C03619=1072.595,223.808,-82.460,174.049,27.815,154.953
C03620=1072.590,223.559,-82.434,174.047,27.812,154.952
C03621=1072.583,223.310,-82.409,174.044,27.808,154.952
C03622=1072.578,223.061,-82.383,174.043,27.804,154.951
C03623=1072.572,222.850,-82.361,174.041,27.800,154.951
C03624=1072.568,222.638,-82.338,174.039,27.797,154.950
C03625=1072.563,222.426,-82.317,174.037,27.794,154.949
C03626=1072.558,222.213,-82.294,174.035,27.790,154.949
C03627=1072.553,222.002,-82.272,174.033,27.787,154.948
C03628=1072.548,221.790,-82.250,174.032,27.784,154.948
C03629=1072.543,221.577,-82.228,174.030,27.780,154.947
C03630=1072.538,221.365,-82.207,174.028,27.777,154.947
C03631=1072.533,221.116,-82.181,174.025,27.773,154.946
C03632=1072.526,220.868,-82.155,174.023,27.769,154.946
C03633=1072.520,220.619,-82.129,174.022,27.766,154.945
C03634=1072.515,220.371,-82.104,174.019,27.761,154.944
C03635=1072.509,220.122,-82.078,174.017,27.758,154.944
C03636=1072.503,219.873,-82.052,174.015,27.754,154.943
C03637=1072.497,219.625,-82.027,174.012,27.750,154.943
C03638=1072.491,219.377,-82.001,174.010,27.746,154.942
C03639=1072.485,219.128,-81.975,174.009,27.743,154.941
C03640=1072.479,218.879,-81.950,174.006,27.738,154.941
C03641=1072.473,218.630,-81.924,174.004,27.734,154.940
C03642=1072.468,218.382,-81.899,174.002,27.731,154.940
C03643=1072.462,218.133,-81.873,173.999,27.727,154.939
C03644=1072.456,217.885,-81.848,173.998,27.723,154.938
C03645=1072.450,217.636,-81.822,173.996,27.719,154.938
C03646=1072.444,217.387,-81.796,173.994,27.715,154.937
C03647=1072.439,217.139,-81.771,173.991,27.711,154.936
C03648=1072.433,216.890,-81.746,173.989,27.707,154.936
C03649=1072.427,216.641,-81.720,173.987,27.703,154.935
C03650=1072.421,216.393,-81.695,173.985,27.699,154.935
C03651=1072.415,216.144,-81.669,173.983,27.695,154.934
C03652=1072.410,215.896,-81.644,173.981,27.692,154.933
C03653=1072.404,215.647,-81.618,173.978,27.688,154.933
C03654=1072.398,215.398,-81.593,173.976,27.684,154.932
C03655=1072.392,215.149,-81.567,173.975,27.680,154.931
C03656=1072.386,214.901,-81.542,173.972,27.676,154.931
C03657=1072.381,214.652,-81.518,173.970,27.672,154.930
C03658=1072.375,214.403,-81.492,173.968,27.668,154.930
C03659=1072.369,214.154,-81.466,173.965,27.664,154.929
C03660=1072.363,213.906,-81.441,173.964,27.660,154.928
C03661=1072.358,213.657,-81.415,173.962,27.656,154.928
C03662=1072.352,213.409,-81.390,173.960,27.652,154.927
C03663=1072.346,213.161,-81.365,173.957,27.648,154.926
C03664=1072.340,212.912,-81.340,173.956,27.645,154.926
C03665=1072.335,212.663,-81.315,173.954,27.641,154.925
C03666=1072.328,212.414,-81.289,173.951,27.637,154.925
C03667=1072.323,212.166,-81.264,173.949,27.633,154.924
C03668=1072.317,211.917,-81.240,173.947,27.629,154.923
C03669=1072.311,211.668,-81.214,173.945,27.625,154.923
C03670=1072.306,211.420,-81.189,173.943,27.621,154.922
C03671=1072.300,211.171,-81.163,173.941,27.617,154.922
C03672=1072.294,210.922,-81.139,173.939,27.613,154.921
C03673=1072.288,210.673,-81.113,173.937,27.609,154.920
C03674=1072.282,210.425,-81.088,173.935,27.606,154.920
C03675=1072.276,210.176,-81.064,173.933,27.602,154.919
C03676=1072.270,209.927,-81.038,173.930,27.598,154.918
C03677=1072.264,209.679,-81.013,173.928,27.593,154.918
C03678=1072.258,209.430,-80.989,173.927,27.590,154.917
C03679=1072.249,209.010,-80.946,173.923,27.583,154.916
C03680=1072.239,208.591,-80.904,173.919,27.577,154.915
C03681=1072.229,208.171,-80.862,173.916,27.570,154.914
C03682=1072.220,207.751,-80.820,173.912,27.563,154.913
C03683=1072.195,206.710,-80.719,173.782,27.496,154.911
C03684=1072.190,206.461,-80.694,173.780,27.493,154.911
C03685=1072.184,206.212,-80.670,173.778,27.490,154.911
C03686=1072.178,205.964,-80.646,173.776,27.487,154.910
C03687=1072.173,205.715,-80.622,173.773,27.484,154.910
C03688=1072.167,205.466,-80.597,173.771,27.480,154.909
C03689=1072.161,205.217,-80.573,173.769,27.477,154.909
C03690=1072.155,204.969,-80.549,173.767,27.475,154.909
C03691=1072.150,204.720,-80.525,173.765,27.472,154.908
C03692=1072.144,204.471,-80.500,173.762,27.469,154.908
C03693=1072.139,204.222,-80.476,173.760,27.465,154.907
C03694=1072.133,203.974,-80.452,173.758,27.463,154.907
C03695=1072.127,203.724,-80.428,173.756,27.460,154.907
C03696=1072.122,203.476,-80.404,173.753,27.457,154.906
C03697=1072.116,203.227,-80.381,173.751,27.454,154.906
C03698=1072.111,202.979,-80.356,173.749,27.451,154.905
C03699=1072.105,202.729,-80.332,173.747,27.448,154.905
C03700=1072.099,202.481,-80.307,173.745,27.444,154.905
C03701=1072.094,202.232,-80.284,173.742,27.441,154.904
C03702=1072.088,201.983,-80.260,173.741,27.439,154.904
C03703=1072.082,201.734,-80.236,173.738,27.436,154.903
C03704=1072.076,201.486,-80.212,173.736,27.433,154.903
C03705=1072.070,201.238,-80.188,173.733,27.430,154.903
C03706=1072.065,200.988,-80.164,173.732,27.427,154.902
C03707=1072.059,200.739,-80.141,173.729,27.424,154.902
C03708=1072.053,200.491,-80.117,173.727,27.421,154.902
C03709=1072.047,200.241,-80.093,173.724,27.418,154.901
C03710=1072.041,199.993,-80.069,173.723,27.416,154.901
C03711=1072.036,199.744,-80.045,173.720,27.413,154.900
C03712=1072.030,199.495,-80.022,173.718,27.410,154.900
C03713=1072.024,199.246,-79.998,173.716,27.407,154.900
C03714=1072.018,198.998,-79.974,173.714,27.404,154.899
C03715=1072.013,198.749,-79.950,173.712,27.401,154.899
C03716=1072.007,198.500,-79.927,173.709,27.398,154.898
C03717=1072.001,198.251,-79.903,173.707,27.395,154.898
C03718=1071.996,198.002,-79.879,173.705,27.393,154.898
C03719=1071.989,197.754,-79.856,173.703,27.390,154.897
C03720=1071.984,197.505,-79.832,173.700,27.387,154.897
C03721=1071.978,197.256,-79.808,173.699,27.384,154.897
C03722=1071.972,197.007,-79.784,173.696,27.381,154.896
C03723=1071.967,196.758,-79.761,173.694,27.378,154.896
C03724=1071.961,196.510,-79.737,173.692,27.375,154.895
C03725=1071.956,196.261,-79.714,173.690,27.372,154.895
C03726=1071.950,196.012,-79.690,173.688,27.369,154.895
C03727=1071.943,195.763,-79.667,173.685,27.366,154.894
C03728=1071.938,195.514,-79.642,173.684,27.364,154.894
C03729=1071.932,195.265,-79.619,173.681,27.361,154.893
C03730=1071.927,195.017,-79.595,173.679,27.358,154.893
C03731=1071.921,194.768,-79.572,173.677,27.355,154.893
C03732=1071.915,194.520,-79.549,173.675,27.352,154.892
C03733=1071.910,194.270,-79.525,173.672,27.349,154.892
C03734=1071.904,194.021,-79.501,173.671,27.346,154.892
C03735=1071.898,193.773,-79.478,173.668,27.343,154.891
C03736=1071.893,193.523,-79.454,173.666,27.340,154.891
C03737=1071.887,193.275,-79.431,173.664,27.337,154.890
C03738=1071.881,193.026,-79.408,173.662,27.334,154.890
C03739=1071.876,192.778,-79.384,173.660,27.331,154.890
C03740=1071.870,192.529,-79.361,173.658,27.328,154.889
C03741=1071.864,192.280,-79.338,173.656,27.325,154.889
C03742=1071.859,192.031,-79.313,173.653,27.323,154.888
C03743=1071.853,191.782,-79.291,173.652,27.320,154.888
C03744=1071.847,191.501,-79.264,173.649,27.317,154.888
C03745=1071.841,191.219,-79.238,173.647,27.314,154.887
C03746=1071.834,190.938,-79.211,173.645,27.310,154.887
C03747=1071.828,190.656,-79.184,173.642,27.307,154.886
C03748=1071.822,190.407,-79.161,173.640,27.304,154.886
C03749=1071.817,190.158,-79.138,173.637,27.301,154.886
C03750=1071.811,189.909,-79.115,173.636,27.298,154.885
C03751=1071.805,189.661,-79.091,173.633,27.295,154.885
C03752=1071.800,189.411,-79.068,173.631,27.292,154.884
C03753=1071.795,189.162,-79.045,173.629,27.289,154.884
C03754=1071.789,188.914,-79.022,173.627,27.286,154.884
C03755=1071.783,188.665,-78.998,173.625,27.283,154.883
C03756=1071.778,188.416,-78.975,173.623,27.281,154.883
C03757=1071.772,188.167,-78.952,173.621,27.278,154.882
C03758=1071.766,187.918,-78.929,173.619,27.275,154.882
C03759=1071.761,187.669,-78.905,173.617,27.272,154.882
C03760=1071.755,187.421,-78.881,173.614,27.269,154.881
C03761=1071.750,187.172,-78.859,173.613,27.267,154.881
C03762=1071.744,186.923,-78.836,173.610,27.263,154.881
C03763=1071.739,186.674,-78.812,173.608,27.260,154.880
C03764=1071.733,186.425,-78.789,173.606,27.258,154.880
C03765=1071.728,186.176,-78.766,173.604,27.255,154.879
C03766=1071.722,185.927,-78.743,173.602,27.252,154.879
C03767=1071.717,185.678,-78.720,173.600,27.249,154.879
C03768=1071.711,185.429,-78.697,173.598,27.246,154.878
C03769=1071.705,185.180,-78.674,173.596,27.243,154.878
C03770=1071.700,184.931,-78.651,173.594,27.240,154.877
C03771=1071.694,184.683,-78.628,173.592,27.237,154.877
C03772=1071.688,184.433,-78.605,173.590,27.234,154.877
C03773=1071.682,184.185,-78.582,173.587,27.232,154.876
C03774=1071.677,183.936,-78.559,173.586,27.229,154.876
C03775=1071.671,183.687,-78.536,173.583,27.226,154.875
C03776=1071.665,183.438,-78.513,173.582,27.224,154.875
C03777=1071.659,183.189,-78.490,173.579,27.221,154.875
C03778=1071.653,182.940,-78.468,173.577,27.218,154.874
C03779=1071.647,182.691,-78.445,173.575,27.215,154.874
C03780=1071.642,182.443,-78.422,173.573,27.212,154.874
C03781=1071.636,182.194,-78.399,173.571,27.210,154.873
C03782=1071.630,181.945,-78.376,173.569,27.207,154.873
C03783=1071.624,181.696,-78.354,173.567,27.204,154.873
C03784=1071.618,181.447,-78.331,173.565,27.201,154.872
C03785=1071.612,181.198,-78.309,173.563,27.198,154.872
C03786=1071.607,180.949,-78.286,173.561,27.196,154.872
C03787=1071.602,180.701,-78.263,173.559,27.193,154.871
C03788=1071.595,180.452,-78.241,173.557,27.190,154.871
C03789=1071.589,180.203,-78.218,173.555,27.188,154.871
C03790=1071.584,179.954,-78.195,173.552,27.185,154.870
C03791=1071.578,179.705,-78.173,173.551,27.182,154.870
C03792=1071.573,179.456,-78.150,173.548,27.179,154.869
C03793=1071.566,179.207,-78.127,173.547,27.177,154.869
C03794=1071.560,178.958,-78.104,173.544,27.174,154.869
C03795=1071.555,178.709,-78.081,173.543,27.171,154.868
C03796=1071.549,178.460,-78.059,173.540,27.168,154.868
C03797=1071.543,178.211,-78.037,173.539,27.166,154.868
C03798=1071.537,177.962,-78.014,173.536,27.163,154.867
C03799=1071.532,177.714,-77.992,173.534,27.160,154.867
C03800=1071.526,177.465,-77.969,173.532,27.157,154.867
C03801=1071.520,177.216,-77.947,173.530,27.154,154.866
C03802=1071.514,176.967,-77.924,173.529,27.152,154.866
C03803=1071.509,176.718,-77.902,173.526,27.148,154.865
C03804=1071.503,176.469,-77.879,173.525,27.146,154.865
C03805=1071.497,176.220,-77.856,173.522,27.143,154.865
C03806=1071.492,175.971,-77.834,173.521,27.140,154.864
C03807=1071.486,175.723,-77.811,173.518,27.137,154.864
C03808=1071.479,175.441,-77.786,173.516,27.134,154.864
C03809=1071.473,175.158,-77.761,173.513,27.131,154.863
C03810=1071.466,174.877,-77.735,173.512,27.129,154.863
C03811=1071.460,174.595,-77.710,173.510,27.125,154.862
C03812=1071.454,174.345,-77.688,173.507,27.122,154.862
C03813=1071.448,174.096,-77.665,173.506,27.120,154.862
C03814=1071.444,173.847,-77.643,173.503,27.117,154.861
C03815=1071.437,173.599,-77.620,173.502,27.114,154.861
C03816=1071.431,173.350,-77.597,173.499,27.111,154.861
C03817=1071.426,173.100,-77.575,173.498,27.109,154.860
C03818=1071.420,172.852,-77.553,173.495,27.106,154.860
C03819=1071.415,172.603,-77.531,173.494,27.103,154.859
C03820=1071.409,172.354,-77.508,173.491,27.100,154.859
C03821=1071.403,172.105,-77.486,173.490,27.097,154.859
C03822=1071.398,171.857,-77.464,173.488,27.094,154.858
C03823=1071.392,171.607,-77.442,173.486,27.092,154.858
C03824=1071.386,171.359,-77.419,173.484,27.089,154.858
C03825=1071.380,171.109,-77.397,173.482,27.086,154.857
C03826=1071.375,170.860,-77.375,173.480,27.083,154.857
C03827=1071.369,170.612,-77.353,173.478,27.081,154.856
C03828=1071.364,170.362,-77.331,173.476,27.078,154.856
C03829=1071.358,170.113,-77.308,173.474,27.075,154.856
C03830=1071.352,169.865,-77.286,173.472,27.072,154.855
C03831=1071.347,169.616,-77.263,173.470,27.069,154.855
C03832=1071.341,169.366,-77.241,173.468,27.066,154.855
C03833=1071.336,169.118,-77.220,173.466,27.064,154.854
C03834=1071.330,168.869,-77.197,173.464,27.061,154.854
C03835=1071.324,168.619,-77.175,173.463,27.058,154.853
C03836=1071.319,168.371,-77.154,173.460,27.055,154.853
C03837=1071.313,168.122,-77.131,173.459,27.052,154.853
C03838=1071.308,167.872,-77.108,173.456,27.050,154.852
C03839=1071.302,167.624,-77.087,173.455,27.047,154.852
C03840=1071.296,167.375,-77.064,173.452,27.044,154.852
C03841=1071.290,167.126,-77.042,173.451,27.041,154.851
C03842=1071.285,166.877,-77.021,173.448,27.038,154.851
C03843=1071.280,166.628,-76.998,173.447,27.036,154.851
C03844=1071.274,166.380,-76.976,173.445,27.033,154.850
C03845=1071.269,166.130,-76.954,173.443,27.030,154.850
C03846=1071.263,165.881,-76.933,173.442,27.027,154.849
C03847=1071.258,165.632,-76.911,173.439,27.024,154.849
C03848=1071.252,165.383,-76.888,173.438,27.022,154.849
C03849=1071.246,165.135,-76.866,173.435,27.019,154.848
C03850=1071.241,164.885,-76.844,173.434,27.016,154.848
C03851=1071.235,164.636,-76.823,173.431,27.013,154.848
C03852=1071.230,164.387,-76.801,173.430,27.010,154.847
C03853=1071.224,164.138,-76.778,173.428,27.008,154.847
C03854=1071.219,163.890,-76.757,173.426,27.005,154.846
C03855=1071.213,163.640,-76.734,173.424,27.002,154.846
C03856=1071.208,163.392,-76.713,173.422,26.999,154.846
C03857=1071.202,163.142,-76.691,173.421,26.997,154.845
C03858=1071.197,162.894,-76.670,173.418,26.994,154.845
C03859=1071.191,162.645,-76.647,173.417,26.991,154.844
C03860=1071.186,162.395,-76.624,173.415,26.988,154.844
C03861=1071.180,162.147,-76.603,173.413,26.985,154.844
C03862=1071.175,161.897,-76.581,173.411,26.983,154.843
C03863=1071.169,161.649,-76.560,173.409,26.980,154.843
C03864=1071.164,161.399,-76.537,173.407,26.977,154.843
C03865=1071.158,161.151,-76.516,173.405,26.974,154.842
C03866=1071.152,160.902,-76.494,173.403,26.972,154.842
C03867=1071.147,160.653,-76.473,173.402,26.969,154.841
C03868=1071.141,160.404,-76.451,173.400,26.966,154.841
C03869=1071.135,160.154,-76.429,173.398,26.963,154.841
C03870=1071.129,159.906,-76.408,173.396,26.960,154.840
C03871=1071.124,159.656,-76.386,173.394,26.958,154.840
C03872=1071.117,159.374,-76.361,173.392,26.955,154.840
C03873=1071.111,159.092,-76.337,173.389,26.951,154.839
C03874=1071.104,158.810,-76.313,173.388,26.949,154.839
C03875=1071.098,158.527,-76.289,173.386,26.946,154.838
C03876=1071.092,158.278,-76.266,173.384,26.943,154.838
C03877=1071.087,158.029,-76.245,173.382,26.940,154.838
C03878=1071.080,157.780,-76.224,173.380,26.937,154.837
C03879=1071.075,157.531,-76.202,173.378,26.934,154.837
C03880=1071.069,157.282,-76.180,173.376,26.932,154.837
C03881=1071.064,157.033,-76.159,173.375,26.929,154.836
C03882=1071.058,156.784,-76.137,173.372,26.926,154.836
C03883=1071.052,156.535,-76.117,173.371,26.924,154.836
C03884=1071.046,156.286,-76.095,173.369,26.920,154.835
C03885=1071.042,156.037,-76.073,173.367,26.918,154.835
C03886=1071.035,155.788,-76.051,173.366,26.915,154.834
C03887=1071.030,155.539,-76.030,173.363,26.912,154.834
C03888=1071.024,155.290,-76.009,173.362,26.910,154.834
C03889=1071.018,155.041,-75.988,173.359,26.907,154.833
C03890=1071.012,154.792,-75.966,173.358,26.904,154.833
C03891=1071.007,154.543,-75.945,173.356,26.902,154.833
C03892=1071.000,154.294,-75.923,173.354,26.899,154.832
C03893=1070.996,154.045,-75.902,173.352,26.896,154.832
C03894=1070.990,153.795,-75.881,173.351,26.893,154.832
C03895=1070.984,153.547,-75.859,173.348,26.891,154.831
C03896=1070.978,153.298,-75.838,173.347,26.888,154.831
C03897=1070.973,153.049,-75.817,173.345,26.885,154.830
C03898=1070.967,152.799,-75.796,173.343,26.883,154.830
C03899=1070.961,152.551,-75.774,173.342,26.880,154.830
C03900=1070.955,152.302,-75.753,173.339,26.877,154.829
C03901=1070.950,152.053,-75.732,173.338,26.875,154.829
C03902=1070.944,151.804,-75.711,173.336,26.872,154.829
C03903=1070.938,151.555,-75.689,173.334,26.869,154.828
C03904=1070.933,151.306,-75.669,173.332,26.866,154.828
C03905=1070.927,151.056,-75.647,173.331,26.864,154.828
C03906=1070.921,150.808,-75.626,173.328,26.861,154.827
C03907=1070.915,150.558,-75.605,173.327,26.858,154.827
C03908=1070.910,150.310,-75.584,173.324,26.855,154.827
C03909=1070.904,150.061,-75.563,173.323,26.853,154.826
C03910=1070.898,149.811,-75.541,173.322,26.850,154.826
C03911=1070.893,149.563,-75.520,173.319,26.847,154.826
C03912=1070.887,149.313,-75.499,173.318,26.844,154.825
C03913=1070.881,149.064,-75.478,173.316,26.842,154.825
C03914=1070.876,148.815,-75.457,173.314,26.839,154.824
C03915=1070.870,148.566,-75.436,173.312,26.836,154.824
C03916=1070.864,148.317,-75.415,173.311,26.834,154.824
C03917=1070.858,148.068,-75.394,173.308,26.830,154.823
C03918=1070.853,147.819,-75.373,173.307,26.828,154.823
C03919=1070.847,147.570,-75.352,173.305,26.825,154.823
C03920=1070.842,147.320,-75.331,173.303,26.823,154.822
C03921=1070.836,147.072,-75.310,173.301,26.820,154.822
C03922=1070.829,146.822,-75.289,173.300,26.817,154.821
C03923=1070.824,146.574,-75.268,173.298,26.815,154.821
C03924=1070.819,146.325,-75.247,173.296,26.812,154.821
C03925=1070.813,146.076,-75.226,173.295,26.809,154.820
C03926=1070.807,145.826,-75.205,173.292,26.807,154.820
C03927=1070.802,145.578,-75.184,173.291,26.804,154.820
C03928=1070.795,145.328,-75.164,173.289,26.801,154.819
C03929=1070.790,145.079,-75.143,173.287,26.799,154.819
C03930=1070.784,144.830,-75.121,173.285,26.796,154.819
C03931=1070.778,144.581,-75.101,173.284,26.793,154.818
C03932=1070.773,144.332,-75.080,173.281,26.790,154.818
C03933=1070.766,144.083,-75.059,173.280,26.788,154.818
C03934=1070.761,143.834,-75.039,173.279,26.785,154.817
C03935=1070.755,143.585,-75.017,173.276,26.782,154.817
C03936=1070.749,143.302,-74.994,173.275,26.779,154.816
C03937=1070.742,143.020,-74.970,173.272,26.776,154.816
C03938=1070.736,142.737,-74.947,173.271,26.773,154.816
C03939=1070.729,142.455,-74.923,173.269,26.770,154.815
C03940=1070.724,142.205,-74.902,173.267,26.767,154.815
C03941=1070.718,141.956,-74.882,173.265,26.765,154.815
C03942=1070.712,141.707,-74.861,173.263,26.762,154.814
C03943=1070.707,141.458,-74.840,173.262,26.759,154.814
C03944=1070.702,141.209,-74.820,173.259,26.756,154.813
C03945=1070.696,140.959,-74.799,173.258,26.754,154.813
C03946=1070.689,140.711,-74.778,173.256,26.751,154.813
C03947=1070.684,140.462,-74.758,173.255,26.748,154.812
C03948=1070.679,140.213,-74.737,173.252,26.746,154.812
C03949=1070.672,139.963,-74.717,173.251,26.743,154.812
C03950=1070.667,139.715,-74.695,173.250,26.740,154.811
C03951=1070.661,139.466,-74.675,173.247,26.737,154.811
C03952=1070.655,139.216,-74.655,173.246,26.735,154.811
C03953=1070.650,138.967,-74.634,173.244,26.732,154.810
C03954=1070.644,138.718,-74.613,173.243,26.730,154.810
C03955=1070.638,138.469,-74.593,173.240,26.726,154.809
C03956=1070.632,138.220,-74.572,173.239,26.724,154.809
C03957=1070.626,137.971,-74.552,173.237,26.721,154.809
C03958=1070.621,137.722,-74.531,173.235,26.718,154.808
C03959=1070.616,137.473,-74.511,173.234,26.716,154.808
C03960=1070.609,137.223,-74.490,173.232,26.713,154.808
C03961=1070.604,136.974,-74.470,173.231,26.710,154.807
C03962=1070.598,136.725,-74.450,173.228,26.707,154.807
C03963=1070.593,136.476,-74.429,173.227,26.705,154.807
C03964=1070.586,136.227,-74.408,173.225,26.702,154.806
C03965=1070.580,135.978,-74.388,173.223,26.699,154.806
C03966=1070.575,135.729,-74.367,173.221,26.697,154.806
C03967=1070.569,135.480,-74.347,173.220,26.694,154.805
C03968=1070.564,135.231,-74.327,173.218,26.691,154.805
C03969=1070.557,134.982,-74.306,173.216,26.689,154.805
C03970=1070.552,134.733,-74.286,173.215,26.686,154.804
C03971=1070.546,134.484,-74.266,173.213,26.683,154.804
C03972=1070.541,134.235,-74.245,173.212,26.681,154.803
C03973=1070.535,133.986,-74.225,173.209,26.678,154.803
C03974=1070.529,133.736,-74.204,173.208,26.675,154.803
C03975=1070.523,133.487,-74.185,173.206,26.673,154.802
C03976=1070.518,133.238,-74.164,173.205,26.670,154.802
C03977=1070.512,132.989,-74.144,173.202,26.667,154.802
C03978=1070.506,132.740,-74.123,173.201,26.665,154.801
C03979=1070.500,132.491,-74.103,173.199,26.662,154.801
C03980=1070.495,132.242,-74.083,173.198,26.659,154.800
C03981=1070.489,131.992,-74.063,173.196,26.656,154.800
C03982=1070.484,131.743,-74.043,173.194,26.654,154.800
C03983=1070.478,131.494,-74.023,173.193,26.651,154.799
C03984=1070.472,131.245,-74.003,173.191,26.649,154.799
C03985=1070.466,130.996,-73.982,173.189,26.646,154.799
C03986=1070.460,130.747,-73.962,173.187,26.643,154.798
C03987=1070.454,130.498,-73.942,173.186,26.640,154.798
C03988=1070.448,130.249,-73.922,173.184,26.638,154.798
C03989=1070.443,129.999,-73.902,173.182,26.635,154.797
C03990=1070.437,129.751,-73.882,173.180,26.632,154.797
C03991=1070.430,129.501,-73.862,173.179,26.630,154.797
C03992=1070.424,129.252,-73.842,173.178,26.627,154.796
C03993=1070.419,129.003,-73.821,173.175,26.624,154.796
C03994=1070.413,128.754,-73.802,173.174,26.622,154.796
C03995=1070.407,128.505,-73.782,173.172,26.619,154.795
C03996=1070.401,128.256,-73.762,173.171,26.617,154.795
C03997=1070.396,128.006,-73.741,173.168,26.614,154.795
C03998=1070.390,127.757,-73.721,173.167,26.611,154.794
C03999=1070.384,127.508,-73.702,173.165,26.609,154.794
C04000=1070.378,127.226,-73.679,173.163,26.606,154.793
C04001=1070.371,126.943,-73.656,173.162,26.602,154.793
C04002=1070.364,126.660,-73.634,173.159,26.599,154.793
C04003=1070.358,126.377,-73.611,173.158,26.596,154.792
C04004=1070.352,126.128,-73.591,173.156,26.594,154.792
C04005=1070.346,125.879,-73.572,173.154,26.591,154.792
C04006=1070.340,125.630,-73.552,173.153,26.588,154.791
C04007=1070.335,125.380,-73.532,173.151,26.586,154.791
C04008=1070.329,125.132,-73.512,173.150,26.583,154.790
C04009=1070.323,124.883,-73.492,173.148,26.580,154.790
C04010=1070.317,124.633,-73.473,173.146,26.578,154.790
C04011=1070.311,124.385,-73.453,173.144,26.575,154.789
C04012=1070.306,124.134,-73.432,173.143,26.572,154.789
C04013=1070.300,123.885,-73.412,173.141,26.570,154.789
C04014=1070.294,123.636,-73.392,173.140,26.567,154.788
C04015=1070.288,123.387,-73.373,173.138,26.564,154.788
C04016=1070.282,123.138,-73.353,173.136,26.562,154.788
C04017=1070.277,122.888,-73.333,173.135,26.559,154.787
C04018=1070.271,122.640,-73.313,173.133,26.556,154.787
C04019=1070.265,122.391,-73.294,173.131,26.553,154.787
C04020=1070.260,122.141,-73.274,173.129,26.551,154.786
C04021=1070.254,121.893,-73.254,173.128,26.548,154.786
C04022=1070.248,121.643,-73.235,173.126,26.545,154.785
C04023=1070.243,121.394,-73.215,173.125,26.543,154.785
C04024=1070.237,121.145,-73.195,173.123,26.540,154.785
C04025=1070.231,120.896,-73.175,173.121,26.537,154.784
C04026=1070.225,120.646,-73.156,173.120,26.534,154.784
C04027=1070.219,120.398,-73.136,173.118,26.532,154.784
C04028=1070.214,120.148,-73.117,173.117,26.529,154.783
C04029=1070.208,119.899,-73.096,173.115,26.526,154.783
C04030=1070.203,119.650,-73.077,173.113,26.523,154.782
C04031=1070.197,119.401,-73.057,173.112,26.521,154.782
C04032=1070.191,119.151,-73.038,173.110,26.518,154.782
C04033=1070.185,118.903,-73.018,173.109,26.516,154.781
C04034=1070.180,118.654,-72.999,173.107,26.513,154.781
C04035=1070.174,118.405,-72.979,173.105,26.510,154.781
C04036=1070.168,118.156,-72.960,173.103,26.507,154.780
C04037=1070.163,117.906,-72.940,173.102,26.505,154.780
C04038=1070.157,117.657,-72.920,173.100,26.502,154.780
C04039=1070.151,117.408,-72.901,173.099,26.499,154.779
C04040=1070.146,117.159,-72.881,173.098,26.496,154.779
C04041=1070.140,116.909,-72.862,173.095,26.493,154.778
C04042=1070.134,116.660,-72.842,173.094,26.491,154.778
C04043=1070.128,116.411,-72.822,173.092,26.488,154.778
C04044=1070.122,116.162,-72.803,173.091,26.485,154.777
C04045=1070.117,115.912,-72.783,173.090,26.482,154.777
C04046=1070.112,115.664,-72.764,173.087,26.480,154.777
C04047=1070.106,115.414,-72.744,173.086,26.477,154.776
C04048=1070.101,115.165,-72.725,173.084,26.474,154.776
C04049=1070.095,114.916,-72.705,173.083,26.471,154.775
C04050=1070.089,114.667,-72.686,173.081,26.469,154.775
C04051=1070.083,114.417,-72.667,173.080,26.466,154.775
C04052=1070.077,114.168,-72.647,173.078,26.463,154.774
C04053=1070.072,113.919,-72.628,173.076,26.460,154.774
C04054=1070.067,113.670,-72.609,173.075,26.458,154.774
C04055=1070.061,113.421,-72.589,173.073,26.455,154.773
C04056=1070.055,113.172,-72.569,173.072,26.452,154.773
C04057=1070.049,112.923,-72.550,173.070,26.450,154.773
C04058=1070.043,112.673,-72.532,173.069,26.447,154.772
C04059=1070.037,112.424,-72.512,173.066,26.444,154.772
C04060=1070.031,112.175,-72.493,173.065,26.442,154.771
C04061=1070.025,111.926,-72.473,173.064,26.439,154.771
C04062=1070.020,111.676,-72.454,173.062,26.436,154.771
C04063=1070.015,111.428,-72.435,173.061,26.433,154.770
C04064=1070.007,111.144,-72.413,173.058,26.430,154.770
C04065=1070.001,110.861,-72.391,173.057,26.427,154.769
C04066=1069.995,110.579,-72.370,173.055,26.424,154.769
C04067=1069.988,110.297,-72.348,173.053,26.421,154.769
C04068=1069.982,110.047,-72.329,173.052,26.419,154.768
C04069=1069.976,109.798,-72.309,173.050,26.416,154.768
C04070=1069.970,109.549,-72.291,173.048,26.413,154.768
C04071=1069.964,109.299,-72.272,173.047,26.410,154.767
C04072=1069.959,109.050,-72.252,173.045,26.408,154.767
C04073=1069.953,108.800,-72.233,173.044,26.405,154.767
C04074=1069.946,108.551,-72.214,173.042,26.402,154.766
C04075=1069.941,108.303,-72.196,173.041,26.400,154.766
C04076=1069.936,108.053,-72.176,173.039,26.397,154.765
C04077=1069.930,107.804,-72.157,173.037,26.394,154.765
C04078=1069.924,107.555,-72.138,173.035,26.392,154.765
C04079=1069.918,107.305,-72.119,173.034,26.389,154.764
C04080=1069.912,107.056,-72.100,173.033,26.386,154.764
C04081=1069.906,106.807,-72.082,173.031,26.383,154.764
C04082=1069.901,106.558,-72.062,173.030,26.381,154.763
C04083=1069.895,106.308,-72.043,173.028,26.378,154.763
C04084=1069.889,106.059,-72.024,173.026,26.375,154.763
C04085=1069.883,105.810,-72.005,173.024,26.373,154.762
C04086=1069.878,105.561,-71.986,173.023,26.370,154.762
C04087=1069.872,105.312,-71.967,173.022,26.367,154.761
C04088=1069.866,105.063,-71.948,173.020,26.364,154.761
C04089=1069.860,104.813,-71.929,173.019,26.362,154.761
C04090=1069.854,104.564,-71.910,173.017,26.359,154.760
C04091=1069.848,104.315,-71.892,173.016,26.356,154.760
C04092=1069.843,104.066,-71.872,173.013,26.354,154.760
C04093=1069.837,103.816,-71.853,173.012,26.351,154.759
C04094=1069.831,103.567,-71.835,173.011,26.348,154.759
C04095=1069.826,103.319,-71.816,173.009,26.345,154.758
C04096=1069.820,103.069,-71.796,173.008,26.343,154.758
C04097=1069.814,102.820,-71.777,173.006,26.340,154.758
C04098=1069.808,102.570,-71.759,173.005,26.337,154.757
C04099=1069.803,102.321,-71.740,173.004,26.335,154.757
C04100=1069.797,102.072,-71.721,173.001,26.332,154.757
C04101=1069.791,101.823,-71.702,173.000,26.329,154.756
C04102=1069.786,101.574,-71.684,172.998,26.326,154.756
C04103=1069.779,101.325,-71.665,172.997,26.324,154.755
C04104=1069.774,101.075,-71.646,172.995,26.321,154.755
C04105=1069.768,100.825,-71.627,172.994,26.318,154.755
C04106=1069.762,100.577,-71.609,172.993,26.316,154.754
C04107=1069.757,100.328,-71.590,172.991,26.313,154.754
C04108=1069.750,100.078,-71.571,172.989,26.310,154.754
C04109=1069.744,99.829,-71.553,172.987,26.307,154.753
C04110=1069.739,99.580,-71.534,172.986,26.305,154.753
C04111=1069.733,99.331,-71.516,172.984,26.302,154.753
C04112=1069.727,99.081,-71.496,172.983,26.299,154.752
C04113=1069.721,98.832,-71.478,172.982,26.297,154.752
C04114=1069.716,98.583,-71.459,172.980,26.294,154.752
C04115=1069.709,98.334,-71.441,172.979,26.291,154.751
C04116=1069.704,98.084,-71.422,172.977,26.289,154.751
C04117=1069.698,97.835,-71.404,172.975,26.286,154.751
C04118=1069.692,97.586,-71.385,172.974,26.283,154.750
C04119=1069.686,97.337,-71.366,172.972,26.281,154.750
C04120=1069.680,97.087,-71.348,172.971,26.278,154.749
C04121=1069.675,96.838,-71.329,172.969,26.275,154.749
C04122=1069.668,96.589,-71.311,172.968,26.272,154.749
C04123=1069.663,96.339,-71.292,172.966,26.270,154.748
C04124=1069.657,96.091,-71.274,172.965,26.267,154.748
C04125=1069.651,95.842,-71.255,172.964,26.264,154.748
C04126=1069.645,95.591,-71.237,172.962,26.262,154.747
C04127=1069.640,95.343,-71.218,172.960,26.259,154.747
C04128=1069.633,95.060,-71.198,172.958,26.256,154.746
C04129=1069.627,94.777,-71.176,172.957,26.253,154.746
C04130=1069.620,94.494,-71.156,172.955,26.250,154.746
C04131=1069.613,94.211,-71.134,172.953,26.247,154.745
C04132=1069.608,93.963,-71.116,172.952,26.244,154.745
C04133=1069.602,93.713,-71.098,172.950,26.242,154.744
C04134=1069.596,93.464,-71.079,172.949,26.239,154.744
C04135=1069.590,93.215,-71.061,172.948,26.236,154.744
C04136=1069.585,92.965,-71.042,172.945,26.233,154.743
C04137=1069.579,92.716,-71.024,172.944,26.231,154.743
C04138=1069.573,92.467,-71.006,172.942,26.228,154.743
C04139=1069.567,92.217,-70.987,172.941,26.225,154.742
C04140=1069.561,91.969,-70.969,172.940,26.222,154.742
C04141=1069.556,91.719,-70.951,172.938,26.220,154.742
C04142=1069.550,91.470,-70.932,172.937,26.217,154.741
C04143=1069.544,91.220,-70.914,172.935,26.214,154.741
C04144=1069.538,90.971,-70.895,172.934,26.211,154.740
C04145=1069.533,90.722,-70.878,172.932,26.209,154.740
C04146=1069.527,90.473,-70.859,172.931,26.206,154.740
C04147=1069.520,90.223,-70.841,172.929,26.203,154.739
C04148=1069.515,89.975,-70.823,172.927,26.201,154.739
C04149=1069.509,89.725,-70.804,172.926,26.198,154.739
C04150=1069.504,89.476,-70.787,172.924,26.195,154.738
C04151=1069.497,89.226,-70.768,172.923,26.193,154.738
C04152=1069.491,88.977,-70.750,172.922,26.190,154.737
C04153=1069.485,88.728,-70.732,172.920,26.187,154.737
C04154=1069.479,88.479,-70.714,172.919,26.185,154.737
C04155=1069.474,88.229,-70.696,172.917,26.182,154.736
C04156=1069.468,87.980,-70.677,172.916,26.179,154.736
C04157=1069.462,87.730,-70.659,172.914,26.177,154.736
C04158=1069.456,87.481,-70.641,172.913,26.174,154.735
C04159=1069.450,87.232,-70.623,172.911,26.171,154.735
C04160=1069.444,86.983,-70.605,172.909,26.168,154.735
C04161=1069.438,86.733,-70.587,172.908,26.166,154.734
C04162=1069.432,86.485,-70.569,172.906,26.163,154.734
C04163=1069.427,86.235,-70.551,172.905,26.160,154.733
C04164=1069.421,85.985,-70.533,172.904,26.158,154.733
C04165=1069.415,85.737,-70.514,172.902,26.155,154.733
C04166=1069.409,85.487,-70.496,172.901,26.152,154.732
C04167=1069.403,85.238,-70.479,172.899,26.150,154.732
C04168=1069.397,84.988,-70.461,172.898,26.147,154.732
C04169=1069.392,84.740,-70.443,172.897,26.144,154.731
C04170=1069.385,84.490,-70.425,172.895,26.141,154.731
C04171=1069.380,84.241,-70.407,172.894,26.139,154.731
C04172=1069.375,83.991,-70.389,172.892,26.136,154.730
C04173=1069.369,83.743,-70.370,172.890,26.133,154.730
C04174=1069.363,83.493,-70.352,172.888,26.130,154.730
C04175=1069.357,83.244,-70.335,172.887,26.128,154.729
C04176=1069.351,82.994,-70.317,172.886,26.125,154.729
C04177=1069.345,82.745,-70.299,172.884,26.122,154.728
C04178=1069.339,82.496,-70.281,172.883,26.120,154.728
C04179=1069.333,82.247,-70.263,172.881,26.117,154.728
C04180=1069.327,81.997,-70.245,172.880,26.114,154.727
C04181=1069.322,81.748,-70.228,172.879,26.111,154.727
C04182=1069.316,81.498,-70.210,172.877,26.109,154.727
C04183=1069.310,81.249,-70.192,172.876,26.106,154.726
C04184=1069.304,81.000,-70.173,172.874,26.103,154.726
C04185=1069.298,80.751,-70.156,172.873,26.100,154.725
C04186=1069.293,80.502,-70.138,172.872,26.098,154.725
C04187=1069.287,80.252,-70.120,172.870,26.095,154.725
C04188=1069.282,80.003,-70.102,172.869,26.092,154.724
C04189=1069.276,79.753,-70.084,172.867,26.089,154.724
C04190=1069.270,79.504,-70.067,172.865,26.087,154.724
C04191=1069.264,79.254,-70.049,172.864,26.084,154.723
C04192=1069.258,78.972,-70.029,172.862,26.081,154.723
C04193=1069.251,78.689,-70.008,172.861,26.078,154.722
C04194=1069.245,78.407,-69.989,172.859,26.074,154.722
C04195=1069.238,78.124,-69.969,172.857,26.072,154.722
C04196=1069.232,77.875,-69.951,172.856,26.069,154.721
C04197=1069.226,77.625,-69.933,172.855,26.066,154.721
C04198=1069.220,77.376,-69.916,172.853,26.064,154.720
C04199=1069.214,77.126,-69.898,172.852,26.061,154.720
C04200=1069.209,76.877,-69.880,172.850,26.058,154.720
C04201=1069.202,76.628,-69.863,172.849,26.056,154.719
C04202=1069.196,76.379,-69.845,172.847,26.053,154.719
C04203=1069.191,76.130,-69.828,172.846,26.050,154.719
C04204=1069.185,75.880,-69.810,172.845,26.048,154.718
C04205=1069.179,75.631,-69.792,172.842,26.044,154.718
C04206=1069.173,75.381,-69.774,172.841,26.042,154.717
C04207=1069.167,75.132,-69.757,172.839,26.039,154.717
C04208=1069.161,74.883,-69.740,172.838,26.036,154.717
C04209=1069.155,74.634,-69.722,172.837,26.034,154.716
C04210=1069.150,74.385,-69.704,172.835,26.031,154.716
C04211=1069.144,74.135,-69.686,172.834,26.028,154.716
C04212=1069.138,73.886,-69.669,172.832,26.026,154.715
C04213=1069.132,73.636,-69.652,172.831,26.023,154.715
C04214=1069.126,73.387,-69.634,172.830,26.020,154.715
C04215=1069.120,73.138,-69.617,172.828,26.018,154.714
C04216=1069.114,72.888,-69.599,172.827,26.015,154.714
C04217=1069.109,72.639,-69.581,172.825,26.012,154.713
C04218=1069.103,72.390,-69.564,172.824,26.010,154.713
C04219=1069.096,72.140,-69.547,172.823,26.007,154.713
C04220=1069.091,71.891,-69.530,172.821,26.004,154.712
C04221=1069.086,71.642,-69.512,172.820,26.001,154.712
C04222=1069.079,71.392,-69.495,172.818,25.999,154.712
C04223=1069.073,71.143,-69.477,172.817,25.996,154.711
C04224=1069.068,70.894,-69.460,172.816,25.993,154.711
C04225=1069.062,70.644,-69.442,172.814,25.991,154.711
C04226=1069.056,70.395,-69.425,172.813,25.988,154.710
C04227=1069.050,70.146,-69.408,172.810,25.985,154.710
C04228=1069.044,69.896,-69.390,172.809,25.982,154.709
C04229=1069.039,69.647,-69.373,172.808,25.979,154.709
C04230=1069.033,69.398,-69.356,172.806,25.977,154.709
C04231=1069.026,69.148,-69.338,172.805,25.974,154.708
C04232=1069.021,68.899,-69.321,172.803,25.971,154.708
C04233=1069.015,68.650,-69.304,172.802,25.969,154.708
C04234=1069.009,68.400,-69.286,172.801,25.966,154.707
C04235=1069.003,68.151,-69.269,172.799,25.963,154.707
C04236=1068.997,67.902,-69.253,172.798,25.961,154.707
C04237=1068.991,67.652,-69.235,172.796,25.958,154.706
C04238=1068.985,67.403,-69.218,172.795,25.955,154.706
C04239=1068.980,67.154,-69.200,172.794,25.952,154.705
C04240=1068.974,66.905,-69.183,172.792,25.950,154.705
C04241=1068.967,66.655,-69.166,172.791,25.947,154.705
C04242=1068.962,66.405,-69.149,172.789,25.944,154.704
C04243=1068.956,66.157,-69.132,172.788,25.942,154.704
C04244=1068.950,65.907,-69.114,172.787,25.939,154.704
C04245=1068.945,65.657,-69.097,172.785,25.936,154.703
C04246=1068.938,65.409,-69.080,172.784,25.934,154.703
C04247=1068.933,65.160,-69.063,172.782,25.931,154.703
C04248=1068.926,64.910,-69.046,172.781,25.928,154.702
C04249=1068.921,64.660,-69.029,172.780,25.926,154.702
C04250=1068.915,64.411,-69.012,172.778,25.923,154.701
C04251=1068.909,64.161,-68.994,172.777,25.920,154.701
C04252=1068.903,63.912,-68.978,172.775,25.917,154.701
C04253=1068.897,63.663,-68.961,172.774,25.915,154.700
C04254=1068.890,63.414,-68.943,172.773,25.912,154.700
C04255=1068.884,63.164,-68.927,172.770,25.909,154.700
C04256=1068.878,62.881,-68.908,172.769,25.906,154.699
C04257=1068.871,62.598,-68.888,172.768,25.903,154.699
C04258=1068.864,62.316,-68.870,172.766,25.901,154.699
C04259=1068.857,62.032,-68.850,172.764,25.897,154.698
C04260=1068.851,61.784,-68.833,172.763,25.894,154.698
C04261=1068.846,61.534,-68.816,172.761,25.892,154.697
C04262=1068.839,61.285,-68.799,172.760,25.889,154.697
C04263=1068.833,61.035,-68.783,172.758,25.886,154.697
C04264=1068.828,60.786,-68.765,172.757,25.884,154.696
C04265=1068.822,60.537,-68.749,172.755,25.881,154.696
C04266=1068.815,60.287,-68.731,172.754,25.879,154.696
C04267=1068.810,60.038,-68.715,172.753,25.876,154.695
C04268=1068.803,59.789,-68.698,172.751,25.873,154.695
C04269=1068.797,59.540,-68.682,172.750,25.871,154.695
C04270=1068.792,59.289,-68.664,172.748,25.868,154.694
C04271=1068.785,59.041,-68.647,172.747,25.865,154.694
C04272=1068.779,58.791,-68.631,172.746,25.863,154.694
C04273=1068.774,58.542,-68.614,172.744,25.860,154.693
C04274=1068.767,58.292,-68.597,172.743,25.858,154.693
C04275=1068.761,58.043,-68.581,172.741,25.855,154.692
C04276=1068.756,57.794,-68.563,172.740,25.852,154.692
C04277=1068.750,57.544,-68.547,172.739,25.850,154.692
C04278=1068.744,57.295,-68.531,172.737,25.847,154.691
C04279=1068.738,57.045,-68.513,172.736,25.844,154.691
C04280=1068.732,56.796,-68.496,172.734,25.842,154.691
C04281=1068.726,56.547,-68.480,172.733,25.839,154.690
C04282=1068.720,56.298,-68.463,172.732,25.836,154.690
C04283=1068.714,56.048,-68.446,172.730,25.834,154.690
C04284=1068.708,55.799,-68.430,172.729,25.831,154.689
C04285=1068.702,55.549,-68.413,172.728,25.828,154.689
C04286=1068.696,55.300,-68.396,172.726,25.825,154.689
C04287=1068.690,55.050,-68.380,172.725,25.823,154.688
C04288=1068.684,54.801,-68.363,172.723,25.820,154.688
C04289=1068.678,54.552,-68.346,172.722,25.817,154.687
C04290=1068.673,54.303,-68.330,172.721,25.815,154.687
C04291=1068.667,54.053,-68.313,172.719,25.812,154.687
C04292=1068.660,53.803,-68.297,172.718,25.809,154.686
C04293=1068.655,53.554,-68.279,172.715,25.806,154.686
C04294=1068.649,53.305,-68.263,172.714,25.803,154.686
C04295=1068.643,53.056,-68.247,172.713,25.801,154.685
C04296=1068.637,52.806,-68.230,172.711,25.798,154.685
C04297=1068.632,52.557,-68.214,172.710,25.795,154.685
C04298=1068.626,52.308,-68.197,172.708,25.793,154.684
C04299=1068.620,52.058,-68.180,172.707,25.790,154.684
C04300=1068.614,51.809,-68.164,172.706,25.787,154.683
C04301=1068.608,51.559,-68.147,172.704,25.785,154.683
C04302=1068.602,51.309,-68.131,172.703,25.782,154.683
C04303=1068.596,51.060,-68.114,172.702,25.779,154.682
C04304=1068.590,50.811,-68.097,172.700,25.777,154.682
C04305=1068.585,50.562,-68.080,172.699,25.774,154.682
C04306=1068.579,50.312,-68.064,172.697,25.771,154.681
C04307=1068.573,50.063,-68.048,172.696,25.768,154.681
C04308=1068.567,49.814,-68.032,172.695,25.766,154.681
C04309=1068.561,49.564,-68.015,172.693,25.763,154.680
C04310=1068.556,49.315,-67.999,172.692,25.760,154.680
C04311=1068.550,49.065,-67.982,172.690,25.758,154.680
C04312=1068.544,48.816,-67.966,172.689,25.755,154.679
C04313=1068.537,48.567,-67.949,172.688,25.752,154.679
C04314=1068.531,48.318,-67.933,172.686,25.750,154.678
C04315=1068.526,48.068,-67.916,172.685,25.747,154.678
C04316=1068.520,47.819,-67.900,172.683,25.744,154.678
C04317=1068.514,47.569,-67.883,172.682,25.741,154.677
C04318=1068.508,47.320,-67.867,172.681,25.739,154.677
C04319=1068.502,47.071,-67.851,172.679,25.736,154.677
C04320=1068.496,46.787,-67.832,172.678,25.733,154.676
C04321=1068.490,46.504,-67.813,172.677,25.730,154.676
C04322=1068.483,46.221,-67.795,172.675,25.726,154.675
C04323=1068.477,45.938,-67.777,172.673,25.723,154.675
C04324=1068.471,45.688,-67.760,172.672,25.721,154.675
C04325=1068.465,45.439,-67.744,172.670,25.718,154.674
C04326=1068.459,45.190,-67.728,172.669,25.715,154.674
C04327=1068.453,44.940,-67.712,172.668,25.712,154.673
C04328=1068.448,44.691,-67.695,172.666,25.710,154.673
C04329=1068.442,44.441,-67.679,172.665,25.707,154.673
C04330=1068.436,44.192,-67.662,172.664,25.704,154.672
C04331=1068.430,43.943,-67.646,172.662,25.702,154.672
C04332=1068.424,43.693,-67.630,172.661,25.699,154.672
C04333=1068.418,43.444,-67.614,172.659,25.696,154.671
C04334=1068.412,43.195,-67.597,172.658,25.693,154.671
C04335=1068.406,42.945,-67.581,172.657,25.691,154.671
C04336=1068.401,42.695,-67.566,172.655,25.688,154.670
C04337=1068.395,42.446,-67.549,172.654,25.685,154.670
C04338=1068.389,42.197,-67.533,172.652,25.683,154.670
C04339=1068.383,41.947,-67.517,172.651,25.680,154.669
C04340=1068.377,41.698,-67.501,172.650,25.677,154.669
C04341=1068.371,41.449,-67.484,172.648,25.675,154.668
C04342=1068.365,41.199,-67.468,172.647,25.672,154.668
C04343=1068.359,40.949,-67.452,172.645,25.670,154.668
C04344=1068.353,40.700,-67.436,172.644,25.667,154.667
C04345=1068.347,40.450,-67.420,172.643,25.664,154.667
C04346=1068.341,40.201,-67.404,172.641,25.662,154.667
C04347=1068.335,39.952,-67.387,172.640,25.659,154.666
C04348=1068.330,39.703,-67.372,172.639,25.656,154.666
C04349=1068.324,39.453,-67.356,172.637,25.654,154.666
C04350=1068.318,39.204,-67.340,172.636,25.651,154.665
C04351=1068.312,38.955,-67.324,172.634,25.648,154.665
C04352=1068.306,38.705,-67.309,172.633,25.645,154.665
C04353=1068.300,38.455,-67.292,172.632,25.643,154.664
C04354=1068.294,38.206,-67.276,172.630,25.640,154.664
C04355=1068.288,37.957,-67.260,172.629,25.637,154.663
C04356=1068.283,37.707,-67.244,172.628,25.634,154.663
C04357=1068.277,37.457,-67.228,172.626,25.632,154.663
C04358=1068.270,37.208,-67.212,172.625,25.629,154.662
C04359=1068.264,36.958,-67.197,172.623,25.627,154.662
C04360=1068.258,36.709,-67.181,172.622,25.624,154.662
C04361=1068.253,36.460,-67.165,172.620,25.622,154.661
C04362=1068.246,36.211,-67.149,172.619,25.619,154.661
C04363=1068.241,35.961,-67.133,172.618,25.616,154.661
C04364=1068.235,35.712,-67.117,172.616,25.614,154.660
C04365=1068.229,35.462,-67.102,172.615,25.611,154.660
C04366=1068.222,35.213,-67.086,172.614,25.608,154.660
C04367=1068.216,34.964,-67.070,172.612,25.606,154.659
C04368=1068.211,34.714,-67.054,172.611,25.603,154.659
C04369=1068.205,34.464,-67.038,172.609,25.600,154.659
C04370=1068.198,34.215,-67.022,172.608,25.597,154.658
C04371=1068.193,33.966,-67.007,172.607,25.595,154.658
C04372=1068.187,33.717,-66.991,172.605,25.592,154.658
C04373=1068.181,33.467,-66.975,172.604,25.590,154.657
C04374=1068.175,33.218,-66.960,172.603,25.587,154.657
C04375=1068.169,32.968,-66.943,172.601,25.585,154.657
C04376=1068.163,32.718,-66.928,172.600,25.582,154.656
C04377=1068.157,32.469,-66.912,172.598,25.579,154.656
C04378=1068.151,32.219,-66.897,172.597,25.577,154.656
C04379=1068.146,31.971,-66.881,172.596,25.574,154.655
C04380=1068.139,31.721,-66.866,172.594,25.571,154.655
C04381=1068.133,31.472,-66.850,172.593,25.568,154.654
C04382=1068.128,31.222,-66.834,172.591,25.566,154.654
C04383=1068.122,30.972,-66.818,172.590,25.563,154.654
C04384=1068.115,30.689,-66.800,172.588,25.560,154.653
C04385=1068.108,30.406,-66.782,172.586,25.557,154.653
C04386=1068.102,30.123,-66.765,172.585,25.554,154.653
C04387=1068.095,29.840,-66.747,172.584,25.551,154.652
C04388=1068.088,29.591,-66.731,172.582,25.548,154.652
C04389=1068.083,29.341,-66.716,172.581,25.546,154.652
C04390=1068.078,29.092,-66.701,172.580,25.543,154.651
C04391=1068.071,28.843,-66.685,172.578,25.540,154.651
C04392=1068.065,28.593,-66.669,172.577,25.538,154.651
C04393=1068.059,28.344,-66.654,172.576,25.535,154.650
C04394=1068.053,28.094,-66.638,172.574,25.533,154.650
C04395=1068.048,27.845,-66.622,172.573,25.530,154.649
C04396=1068.041,27.595,-66.607,172.571,25.528,154.649
C04397=1068.036,27.345,-66.592,172.570,25.525,154.649
C04398=1068.029,27.096,-66.576,172.569,25.522,154.648
C04399=1068.023,26.846,-66.561,172.567,25.519,154.648
C04400=1068.017,26.597,-66.546,172.566,25.517,154.648
C04401=1068.012,26.348,-66.530,172.564,25.514,154.647
C04402=1068.005,26.098,-66.515,172.563,25.512,154.647
C04403=1067.999,25.849,-66.499,172.562,25.509,154.647
C04404=1067.993,25.599,-66.484,172.560,25.507,154.646
C04405=1067.988,25.350,-66.469,172.559,25.504,154.646
C04406=1067.981,25.100,-66.454,172.557,25.501,154.646
C04407=1067.975,24.851,-66.437,172.556,25.498,154.645
C04408=1067.969,24.601,-66.422,172.555,25.496,154.645
C04409=1067.964,24.352,-66.407,172.553,25.493,154.645
C04410=1067.957,24.103,-66.392,172.552,25.491,154.644
C04411=1067.952,23.853,-66.376,172.551,25.488,154.644
C04412=1067.945,23.603,-66.361,172.549,25.486,154.644
C04413=1067.939,23.354,-66.346,172.548,25.483,154.643
C04414=1067.934,23.105,-66.330,172.546,25.480,154.643
C04415=1067.927,22.855,-66.315,172.545,25.478,154.643
C04416=1067.922,22.606,-66.300,172.544,25.475,154.642
C04417=1067.916,22.357,-66.285,172.542,25.472,154.642
C04418=1067.910,22.107,-66.269,172.541,25.470,154.642
C04419=1067.903,21.858,-66.254,172.539,25.467,154.641
C04420=1067.898,21.608,-66.239,172.538,25.465,154.641
C04421=1067.892,21.359,-66.224,172.537,25.462,154.641
C04422=1067.886,21.109,-66.208,172.535,25.460,154.640
C04423=1067.880,20.860,-66.193,172.534,25.457,154.640
C04424=1067.874,20.611,-66.178,172.532,25.454,154.640
C04425=1067.868,20.361,-66.163,172.531,25.451,154.639
C04426=1067.862,20.111,-66.148,172.530,25.449,154.639
C04427=1067.857,19.862,-66.132,172.528,25.447,154.639
C04428=1067.850,19.612,-66.117,172.527,25.444,154.638
C04429=1067.844,19.363,-66.102,172.525,25.441,154.638
C04430=1067.838,19.113,-66.086,172.524,25.439,154.638
C04431=1067.832,18.864,-66.072,172.523,25.436,154.637
C04432=1067.826,18.615,-66.057,172.521,25.433,154.637
C04433=1067.820,18.365,-66.041,172.520,25.431,154.637
C04434=1067.814,18.116,-66.027,172.519,25.428,154.636
C04435=1067.808,17.866,-66.012,172.517,25.426,154.636
C04436=1067.802,17.616,-65.997,172.516,25.423,154.636
C04437=1067.797,17.367,-65.982,172.514,25.421,154.635
C04438=1067.790,17.117,-65.967,172.513,25.418,154.635
C04439=1067.784,16.868,-65.951,172.512,25.415,154.635
C04440=1067.779,16.619,-65.936,172.510,25.413,154.634
C04441=1067.772,16.369,-65.921,172.509,25.410,154.634
C04442=1067.766,16.120,-65.906,172.507,25.408,154.634
C04443=1067.761,15.870,-65.891,172.506,25.405,154.633
C04444=1067.754,15.621,-65.876,172.505,25.402,154.633
C04445=1067.749,15.372,-65.861,172.503,25.400,154.633
C04446=1067.742,15.122,-65.846,172.502,25.397,154.632
C04447=1067.737,14.872,-65.831,172.500,25.395,154.632
C04448=1067.730,14.591,-65.814,172.498,25.392,154.632
C04449=1067.724,14.309,-65.798,172.497,25.389,154.631
C04450=1067.716,14.027,-65.780,172.496,25.386,154.631
C04451=1067.710,13.745,-65.764,172.494,25.383,154.631
C04452=1067.703,13.495,-65.749,172.493,25.381,154.630
C04453=1067.698,13.246,-65.734,172.491,25.378,154.630
C04454=1067.691,12.997,-65.719,172.490,25.375,154.630
C04455=1067.685,12.747,-65.704,172.489,25.373,154.629
C04456=1067.679,12.498,-65.690,172.487,25.371,154.629
C04457=1067.673,12.248,-65.675,172.486,25.368,154.629
C04458=1067.667,11.998,-65.660,172.484,25.365,154.628
C04459=1067.661,11.749,-65.646,172.483,25.363,154.628
C04460=1067.654,11.500,-65.631,172.481,25.360,154.628
C04461=1067.649,11.251,-65.616,172.479,25.357,154.628
C04462=1067.642,11.001,-65.601,172.478,25.355,154.627
C04463=1067.636,10.751,-65.586,172.476,25.353,154.627
C04464=1067.631,10.502,-65.571,172.475,25.350,154.627
C04465=1067.624,10.252,-65.556,172.474,25.348,154.626
C04466=1067.619,10.003,-65.542,172.472,25.345,154.626
C04467=1067.613,9.753,-65.527,172.471,25.342,154.626
C04468=1067.606,9.503,-65.512,172.469,25.340,154.625
C04469=1067.600,9.255,-65.498,172.468,25.338,154.625
C04470=1067.594,9.005,-65.483,172.467,25.335,154.625
C04471=1067.588,8.755,-65.469,172.465,25.332,154.624
C04472=1067.582,8.506,-65.454,172.464,25.330,154.624
C04473=1067.576,8.256,-65.439,172.462,25.327,154.624
C04474=1067.570,8.007,-65.425,172.461,25.325,154.624
C04475=1067.564,7.757,-65.410,172.460,25.322,154.623
C04476=1067.558,7.508,-65.396,172.458,25.319,154.623
C04477=1067.552,7.258,-65.381,172.457,25.317,154.623
C04478=1067.546,7.009,-65.366,172.455,25.315,154.622
C04479=1067.540,6.760,-65.351,172.454,25.312,154.622
C04480=1067.534,6.510,-65.337,172.453,25.310,154.622
C04481=1067.528,6.260,-65.323,172.451,25.307,154.621
C04482=1067.522,6.011,-65.308,172.450,25.304,154.621
C04483=1067.516,5.761,-65.294,172.448,25.302,154.621
C04484=1067.510,5.512,-65.279,172.447,25.300,154.620
C04485=1067.504,5.262,-65.264,172.446,25.297,154.620
C04486=1067.498,5.014,-65.250,172.444,25.294,154.620
C04487=1067.492,4.763,-65.235,172.443,25.292,154.620
C04488=1067.486,4.514,-65.221,172.442,25.289,154.619
C04489=1067.480,4.265,-65.206,172.440,25.287,154.619
C04490=1067.474,4.015,-65.192,172.439,25.284,154.619
C04491=1067.468,3.765,-65.177,172.437,25.282,154.618
C04492=1067.462,3.516,-65.163,172.436,25.279,154.618
C04493=1067.456,3.266,-65.148,172.434,25.277,154.618
C04494=1067.450,3.017,-65.134,172.433,25.274,154.617
C04495=1067.444,2.767,-65.119,172.432,25.272,154.617
C04496=1067.438,2.518,-65.105,172.430,25.269,154.617
C04497=1067.432,2.268,-65.090,172.429,25.267,154.616
C04498=1067.426,2.019,-65.076,172.428,25.264,154.616
C04499=1067.420,1.769,-65.061,172.426,25.262,154.616
C04500=1067.415,1.520,-65.047,172.425,25.259,154.615
C04501=1067.408,1.270,-65.032,172.423,25.256,154.615
C04502=1067.403,1.020,-65.018,172.422,25.254,154.615
C04503=1067.397,0.771,-65.004,172.420,25.252,154.615
C04504=1067.391,0.522,-64.989,172.419,25.249,154.614
C04505=1067.385,0.272,-64.975,172.418,25.246,154.614
C04506=1067.379,0.022,-64.960,172.416,25.244,154.614
C04507=1067.373,-0.227,-64.946,172.415,25.242,154.613
C04508=1067.367,-0.476,-64.932,172.414,25.239,154.613
C04509=1067.361,-0.726,-64.917,172.412,25.236,154.613
C04510=1067.356,-0.975,-64.903,172.411,25.234,154.612
C04511=1067.349,-1.225,-64.889,172.409,25.231,154.612
C04512=1067.342,-1.505,-64.873,172.408,25.229,154.612
C04513=1067.335,-1.785,-64.857,172.407,25.226,154.611
C04514=1067.329,-2.065,-64.841,172.404,25.223,154.611
C04515=1067.322,-2.344,-64.825,172.403,25.220,154.611
C04516=1067.317,-2.594,-64.811,172.402,25.217,154.610
C04517=1067.311,-2.843,-64.796,172.400,25.215,154.610
C04518=1067.305,-3.093,-64.782,172.399,25.213,154.610
C04519=1067.299,-3.342,-64.768,172.398,25.210,154.609
C04520=1067.293,-3.592,-64.753,172.396,25.207,154.609
C04521=1067.287,-3.842,-64.740,172.395,25.205,154.609
C04522=1067.281,-4.091,-64.725,172.393,25.203,154.609
C04523=1067.275,-4.341,-64.711,172.392,25.200,154.608
C04524=1067.268,-4.590,-64.697,172.390,25.198,154.608
C04525=1067.262,-4.840,-64.683,172.389,25.196,154.608
C04526=1067.257,-5.089,-64.669,172.388,25.193,154.607
C04527=1067.250,-5.338,-64.655,172.386,25.190,154.607
C04528=1067.244,-5.588,-64.641,172.385,25.188,154.607
C04529=1067.239,-5.838,-64.627,172.383,25.186,154.607
C04530=1067.232,-6.087,-64.613,172.382,25.183,154.606
C04531=1067.226,-6.337,-64.599,172.380,25.181,154.606
C04532=1067.221,-6.586,-64.585,172.379,25.179,154.606
C04533=1067.214,-6.836,-64.571,172.378,25.176,154.605
C04534=1067.208,-7.085,-64.557,172.376,25.173,154.605
C04535=1067.202,-7.336,-64.543,172.375,25.171,154.605
C04536=1067.196,-7.584,-64.529,172.373,25.169,154.604
C04537=1067.190,-7.834,-64.515,172.372,25.166,154.604
C04538=1067.184,-8.084,-64.501,172.371,25.164,154.604
C04539=1067.178,-8.333,-64.487,172.369,25.161,154.604
C04540=1067.172,-8.582,-64.473,172.368,25.159,154.603
C04541=1067.166,-8.833,-64.458,172.366,25.157,154.603
C04542=1067.160,-9.082,-64.445,172.365,25.154,154.603
C04543=1067.154,-9.331,-64.431,172.364,25.151,154.602
C04544=1067.147,-9.581,-64.417,172.362,25.149,154.602
C04545=1067.142,-9.830,-64.403,172.361,25.147,154.602
C04546=1067.136,-10.080,-64.389,172.359,25.144,154.602
C04547=1067.129,-10.330,-64.376,172.358,25.142,154.601
C04548=1067.124,-10.579,-64.362,172.356,25.140,154.601
C04549=1067.117,-10.828,-64.348,172.355,25.137,154.601
C04550=1067.112,-11.078,-64.334,172.354,25.134,154.600
C04551=1067.106,-11.328,-64.320,172.352,25.132,154.600
C04552=1067.100,-11.577,-64.306,172.350,25.129,154.600
C04553=1067.094,-11.827,-64.292,172.349,25.127,154.600
C04554=1067.087,-12.077,-64.279,172.347,25.125,154.599
C04555=1067.081,-12.326,-64.264,172.346,25.122,154.599
C04556=1067.076,-12.575,-64.250,172.344,25.120,154.599
C04557=1067.070,-12.825,-64.237,172.343,25.118,154.599
C04558=1067.064,-13.075,-64.223,172.341,25.115,154.598
C04559=1067.057,-13.324,-64.210,172.340,25.113,154.598
C04560=1067.052,-13.574,-64.196,172.339,25.111,154.598
C04561=1067.047,-13.823,-64.182,172.337,25.108,154.597
C04562=1067.040,-14.073,-64.168,172.336,25.105,154.597
C04563=1067.034,-14.323,-64.154,172.334,25.103,154.597
C04564=1067.028,-14.571,-64.140,172.333,25.100,154.597
C04565=1067.022,-14.821,-64.127,172.332,25.098,154.596
C04566=1067.015,-15.071,-64.113,172.330,25.096,154.596
C04567=1067.010,-15.321,-64.099,172.329,25.093,154.596
C04568=1067.004,-15.570,-64.086,172.327,25.091,154.595
C04569=1066.998,-15.819,-64.072,172.326,25.089,154.595
C04570=1066.991,-16.069,-64.058,172.324,25.086,154.595
C04571=1066.985,-16.319,-64.045,172.323,25.084,154.595
C04572=1066.980,-16.568,-64.031,172.322,25.082,154.594
C04573=1066.974,-16.817,-64.018,172.320,25.079,154.594
C04574=1066.967,-17.067,-64.004,172.319,25.077,154.594
C04575=1066.961,-17.317,-63.990,172.317,25.075,154.594
C04576=1066.956,-17.544,-63.978,172.316,25.073,154.593
C04577=1066.950,-17.771,-63.966,172.314,25.070,154.593
C04578=1066.945,-17.998,-63.954,172.313,25.068,154.593
C04579=1066.939,-18.226,-63.941,172.312,25.067,154.593
C04580=1066.933,-18.452,-63.929,172.311,25.064,154.592
C04581=1066.928,-18.680,-63.917,172.309,25.062,154.592
C04582=1066.922,-18.906,-63.905,172.308,25.060,154.592
C04583=1066.917,-19.133,-63.893,172.306,25.058,154.592
C04584=1066.911,-19.383,-63.878,172.305,25.055,154.591
C04585=1066.905,-19.633,-63.865,172.304,25.053,154.591
C04586=1066.899,-19.882,-63.852,172.302,25.051,154.591
C04587=1066.893,-20.132,-63.838,172.301,25.048,154.591
C04588=1066.885,-20.454,-63.821,172.298,25.045,154.590
C04589=1066.877,-20.778,-63.803,172.297,25.043,154.590
C04590=1066.869,-21.102,-63.785,172.295,25.039,154.590
C04591=1066.861,-21.425,-63.769,172.294,25.036,154.589
C04592=1066.855,-21.674,-63.755,172.292,25.034,154.589
C04593=1066.850,-21.924,-63.741,172.291,25.032,154.589
C04594=1066.844,-22.173,-63.729,172.289,25.029,154.588
C04595=1066.837,-22.423,-63.716,172.287,25.027,154.588
C04596=1066.832,-22.672,-63.702,172.286,25.024,154.588
C04597=1066.825,-22.922,-63.688,172.284,25.022,154.588
C04598=1066.819,-23.172,-63.675,172.283,25.020,154.588
C04599=1066.814,-23.422,-63.662,172.281,25.018,154.587
C04600=1066.807,-23.671,-63.648,172.280,25.015,154.587
C04601=1066.801,-23.920,-63.635,172.278,25.013,154.587
C04602=1066.796,-24.170,-63.621,172.277,25.011,154.586
C04603=1066.790,-24.419,-63.608,172.275,25.008,154.586
C04604=1066.784,-24.669,-63.595,172.274,25.006,154.586
C04605=1066.777,-24.919,-63.582,172.273,25.004,154.586
C04606=1066.771,-25.169,-63.568,172.271,25.001,154.585
C04607=1066.765,-25.418,-63.555,172.270,24.999,154.585
C04608=1066.759,-25.668,-63.542,172.268,24.997,154.585
C04609=1066.754,-25.917,-63.528,172.267,24.995,154.585
C04610=1066.748,-26.166,-63.515,172.265,24.992,154.584
C04611=1066.742,-26.416,-63.502,172.264,24.990,154.584
C04612=1066.735,-26.666,-63.489,172.263,24.988,154.584
C04613=1066.730,-26.915,-63.475,172.261,24.985,154.584
C04614=1066.724,-27.164,-63.462,172.260,24.983,154.583
C04615=1066.718,-27.414,-63.449,172.258,24.981,154.583
C04616=1066.711,-27.664,-63.436,172.257,24.979,154.583
C04617=1066.705,-27.914,-63.423,172.255,24.976,154.583
C04618=1066.699,-28.163,-63.410,172.254,24.974,154.582
C04619=1066.693,-28.413,-63.397,172.252,24.972,154.582
C04620=1066.687,-28.663,-63.384,172.251,24.970,154.582
C04621=1066.681,-28.912,-63.371,172.249,24.967,154.582
C04622=1066.674,-29.161,-63.358,172.248,24.965,154.581
C04623=1066.668,-29.411,-63.345,172.247,24.963,154.581
C04624=1066.662,-29.660,-63.332,172.245,24.961,154.581
C04625=1066.656,-29.910,-63.319,172.244,24.958,154.581
C04626=1066.651,-30.160,-63.305,172.241,24.956,154.581
C04627=1066.644,-30.410,-63.292,172.240,24.954,154.580
C04628=1066.638,-30.660,-63.279,172.238,24.952,154.580
C04629=1066.632,-30.909,-63.266,172.237,24.949,154.580
C04630=1066.626,-31.159,-63.253,172.235,24.947,154.580
C04631=1066.620,-31.408,-63.240,172.234,24.945,154.579
C04632=1066.614,-31.658,-63.228,172.233,24.943,154.579
C04633=1066.608,-31.907,-63.214,172.231,24.940,154.579
C04634=1066.601,-32.156,-63.201,172.230,24.938,154.579
C04635=1066.596,-32.406,-63.188,172.228,24.936,154.579
C04636=1066.589,-32.656,-63.175,172.227,24.934,154.578
C04637=1066.583,-32.905,-63.163,172.225,24.932,154.578
C04638=1066.577,-33.155,-63.149,172.224,24.930,154.578
C04639=1066.571,-33.405,-63.137,172.222,24.927,154.578
C04640=1066.564,-33.682,-63.123,172.221,24.925,154.577
C04641=1066.558,-33.959,-63.108,172.219,24.922,154.577
C04642=1066.551,-34.236,-63.094,172.217,24.920,154.577
C04643=1066.545,-34.514,-63.079,172.216,24.917,154.577
C04644=1066.539,-34.764,-63.067,172.214,24.915,154.576
C04645=1066.533,-35.014,-63.053,172.213,24.913,154.576
C04646=1066.527,-35.263,-63.041,172.211,24.911,154.576
C04647=1066.520,-35.513,-63.028,172.210,24.908,154.576
C04648=1066.515,-35.763,-63.015,172.208,24.907,154.575
C04649=1066.508,-36.012,-63.002,172.207,24.904,154.575
C04650=1066.502,-36.262,-62.989,172.206,24.902,154.575
C04651=1066.497,-36.512,-62.977,172.204,24.900,154.575
C04652=1066.490,-36.761,-62.963,172.203,24.898,154.574
C04653=1066.484,-37.011,-62.951,172.201,24.895,154.574
C04654=1066.479,-37.259,-62.938,172.199,24.893,154.574
C04655=1066.473,-37.509,-62.925,172.197,24.891,154.574
C04656=1066.467,-37.759,-62.913,172.196,24.888,154.574
C04657=1066.461,-38.008,-62.900,172.194,24.887,154.573
C04658=1066.454,-38.258,-62.888,172.193,24.884,154.573
C04659=1066.448,-38.508,-62.875,172.191,24.882,154.573
C04660=1066.442,-38.757,-62.862,172.190,24.880,154.573
C04661=1066.436,-39.007,-62.849,172.189,24.878,154.572
C04662=1066.430,-39.257,-62.837,172.187,24.876,154.572
C04663=1066.424,-39.506,-62.823,172.186,24.874,154.572
C04664=1066.417,-39.756,-62.811,172.184,24.872,154.572
C04665=1066.411,-40.006,-62.799,172.183,24.869,154.572
C04666=1066.405,-40.255,-62.786,172.181,24.868,154.571
C04667=1066.399,-40.505,-62.773,172.180,24.865,154.571
C04668=1066.393,-40.755,-62.760,172.178,24.863,154.571
C04669=1066.387,-41.004,-62.749,172.177,24.861,154.571
C04670=1066.381,-41.254,-62.736,172.175,24.859,154.571
C04671=1066.375,-41.503,-62.723,172.174,24.857,154.570
C04672=1066.369,-41.753,-62.710,172.172,24.855,154.570
C04673=1066.363,-42.002,-62.699,172.171,24.853,154.570
C04674=1066.357,-42.252,-62.686,172.169,24.851,154.570
C04675=1066.351,-42.501,-62.673,172.168,24.848,154.570
C04676=1066.345,-42.751,-62.660,172.166,24.847,154.569
C04677=1066.338,-43.001,-62.648,172.165,24.844,154.569
C04678=1066.332,-43.251,-62.636,172.162,24.842,154.569
C04679=1066.326,-43.500,-62.623,172.161,24.840,154.569
C04680=1066.320,-43.750,-62.611,172.159,24.838,154.569
C04681=1066.314,-43.999,-62.598,172.158,24.836,154.569
C04682=1066.308,-44.248,-62.586,172.156,24.834,154.568
C04683=1066.302,-44.498,-62.573,172.155,24.832,154.568
C04684=1066.296,-44.748,-62.561,172.154,24.830,154.568
C04685=1066.290,-44.998,-62.549,172.152,24.828,154.568
C04686=1066.284,-45.248,-62.536,172.151,24.825,154.567
C04687=1066.278,-45.498,-62.523,172.149,24.824,154.567
C04688=1066.272,-45.746,-62.511,172.148,24.821,154.567
C04689=1066.265,-45.996,-62.499,172.146,24.819,154.567
C04690=1066.260,-46.246,-62.486,172.145,24.817,154.567
C04691=1066.254,-46.495,-62.474,172.143,24.815,154.566
C04692=1066.247,-46.745,-62.462,172.142,24.813,154.566
C04693=1066.241,-46.995,-62.449,172.140,24.811,154.566
C04694=1066.236,-47.244,-62.437,172.139,24.809,154.566
C04695=1066.229,-47.494,-62.425,172.137,24.807,154.566
C04696=1066.223,-47.744,-62.412,172.136,24.805,154.565
C04697=1066.217,-47.993,-62.400,172.134,24.803,154.565
C04698=1066.211,-48.243,-62.387,172.133,24.801,154.565
C04699=1066.205,-48.492,-62.376,172.131,24.799,154.565
C04700=1066.199,-48.742,-62.363,172.129,24.796,154.565
C04701=1066.194,-48.992,-62.351,172.127,24.795,154.565
C04702=1066.187,-49.242,-62.339,172.126,24.792,154.564
C04703=1066.181,-49.491,-62.326,172.124,24.790,154.564
C04704=1066.175,-49.768,-62.312,172.123,24.788,154.564
C04705=1066.168,-50.047,-62.299,172.121,24.786,154.564
C04706=1066.161,-50.325,-62.285,172.120,24.784,154.563
C04707=1066.154,-50.603,-62.272,172.117,24.782,154.563
C04708=1066.148,-50.852,-62.260,172.116,24.779,154.563
C04709=1066.142,-51.101,-62.248,172.115,24.777,154.563
C04710=1066.136,-51.351,-62.235,172.113,24.776,154.563
C04711=1066.129,-51.601,-62.223,172.111,24.774,154.563
C04712=1066.123,-51.850,-62.211,172.110,24.772,154.563
C04713=1066.117,-52.100,-62.199,172.108,24.770,154.562
C04714=1066.111,-52.349,-62.187,172.107,24.768,154.562
C04715=1066.105,-52.599,-62.174,172.105,24.766,154.562
C04716=1066.098,-52.849,-62.162,172.104,24.764,154.562
C04717=1066.092,-53.099,-62.151,172.102,24.762,154.562
C04718=1066.086,-53.349,-62.139,172.101,24.761,154.562
C04719=1066.080,-53.597,-62.127,172.099,24.758,154.561
C04720=1066.073,-53.847,-62.115,172.098,24.756,154.561
C04721=1066.067,-54.097,-62.103,172.096,24.755,154.561
C04722=1066.061,-54.346,-62.091,172.094,24.752,154.561
C04723=1066.055,-54.596,-62.078,172.092,24.751,154.561
C04724=1066.049,-54.846,-62.067,172.091,24.749,154.561
C04725=1066.042,-55.095,-62.055,172.089,24.747,154.560
C04726=1066.036,-55.345,-62.043,172.088,24.745,154.560
C04727=1066.030,-55.595,-62.031,172.086,24.743,154.560
C04728=1066.024,-55.844,-62.019,172.085,24.741,154.560
C04729=1066.018,-56.094,-62.007,172.083,24.739,154.560
C04730=1066.011,-56.344,-61.995,172.082,24.737,154.560
C04731=1066.005,-56.593,-61.983,172.080,24.735,154.559
C04732=1066.000,-56.843,-61.971,172.078,24.734,154.559
C04733=1065.993,-57.093,-61.960,172.077,24.732,154.559
C04734=1065.987,-57.343,-61.947,172.075,24.729,154.559
C04735=1065.981,-57.592,-61.935,172.074,24.728,154.559
C04736=1065.975,-57.841,-61.924,172.072,24.726,154.559
C04737=1065.969,-58.092,-61.912,172.071,24.724,154.558
C04738=1065.962,-58.341,-61.900,172.069,24.722,154.558
C04739=1065.956,-58.590,-61.888,172.068,24.720,154.558
C04740=1065.950,-58.840,-61.876,172.066,24.719,154.558
C04741=1065.944,-59.090,-61.865,172.065,24.717,154.558
C04742=1065.938,-59.339,-61.853,172.062,24.715,154.558
C04743=1065.931,-59.589,-61.841,172.061,24.713,154.558
C04744=1065.926,-59.839,-61.829,172.059,24.711,154.558
C04745=1065.920,-60.088,-61.818,172.058,24.709,154.557
C04746=1065.913,-60.338,-61.806,172.056,24.707,154.557
C04747=1065.907,-60.588,-61.794,172.055,24.705,154.557
C04748=1065.901,-60.837,-61.782,172.053,24.703,154.557
C04749=1065.895,-61.086,-61.770,172.052,24.701,154.557
C04750=1065.889,-61.337,-61.758,172.050,24.700,154.557
C04751=1065.883,-61.586,-61.747,172.048,24.698,154.556
C04752=1065.877,-61.836,-61.736,172.047,24.696,154.556
C04753=1065.870,-62.086,-61.724,172.045,24.694,154.556
C04754=1065.865,-62.335,-61.711,172.044,24.692,154.556
C04755=1065.858,-62.585,-61.700,172.042,24.690,154.556
C04756=1065.852,-62.835,-61.688,172.041,24.689,154.556
C04757=1065.847,-63.084,-61.677,172.039,24.687,154.556
C04758=1065.840,-63.334,-61.665,172.038,24.685,154.555
C04759=1065.834,-63.583,-61.653,172.036,24.683,154.555
C04760=1065.828,-63.833,-61.642,172.035,24.681,154.555
C04761=1065.822,-64.083,-61.629,172.033,24.680,154.555
C04762=1065.816,-64.332,-61.619,172.031,24.678,154.555
C04763=1065.810,-64.582,-61.607,172.029,24.676,154.555
C04764=1065.804,-64.831,-61.596,172.027,24.674,154.555
C04765=1065.798,-65.081,-61.583,172.026,24.672,154.554
C04766=1065.792,-65.331,-61.572,172.024,24.670,154.554
C04767=1065.785,-65.580,-61.560,172.023,24.668,154.554
C04768=1065.779,-65.860,-61.547,172.021,24.666,154.554
C04769=1065.772,-66.139,-61.534,172.020,24.665,154.554
C04770=1065.766,-66.418,-61.522,172.017,24.662,154.554
C04771=1065.759,-66.697,-61.508,172.016,24.660,154.554
C04772=1065.753,-66.947,-61.497,172.014,24.658,154.553
C04773=1065.746,-67.196,-61.485,172.013,24.656,154.553
C04774=1065.740,-67.446,-61.474,172.011,24.655,154.553
C04775=1065.735,-67.696,-61.462,172.010,24.653,154.553
C04776=1065.728,-67.946,-61.450,172.008,24.652,154.553
C04777=1065.723,-68.195,-61.440,172.006,24.650,154.553
C04778=1065.716,-68.445,-61.428,172.005,24.648,154.553
C04779=1065.710,-68.694,-61.417,172.003,24.646,154.553
C04780=1065.704,-68.944,-61.404,172.002,24.644,154.552
C04781=1065.699,-69.194,-61.393,172.000,24.643,154.552
C04782=1065.692,-69.444,-61.382,171.999,24.641,154.552
C04783=1065.686,-69.693,-61.370,171.997,24.639,154.552
C04784=1065.680,-69.943,-61.359,171.995,24.637,154.552
C04785=1065.675,-70.193,-61.348,171.993,24.635,154.552
C04786=1065.668,-70.442,-61.336,171.992,24.633,154.552
C04787=1065.663,-70.692,-61.325,171.990,24.632,154.552
C04788=1065.657,-70.941,-61.314,171.988,24.630,154.551
C04789=1065.650,-71.191,-61.302,171.987,24.628,154.551
C04790=1065.645,-71.441,-61.291,171.985,24.626,154.551
C04791=1065.639,-71.691,-61.279,171.984,24.625,154.551
C04792=1065.633,-71.940,-61.268,171.982,24.623,154.551
C04793=1065.626,-72.190,-61.257,171.981,24.621,154.551
C04794=1065.621,-72.439,-61.246,171.979,24.619,154.551
C04795=1065.615,-72.689,-61.233,171.977,24.618,154.551
C04796=1065.609,-72.939,-61.222,171.976,24.616,154.550
C04797=1065.603,-73.188,-61.211,171.974,24.614,154.550
C04798=1065.597,-73.438,-61.199,171.973,24.612,154.550
C04799=1065.591,-73.687,-61.188,171.971,24.611,154.550
C04800=1065.585,-73.937,-61.177,171.970,24.609,154.550
C04801=1065.579,-74.187,-61.166,171.968,24.607,154.550
C04802=1065.572,-74.436,-61.154,171.967,24.606,154.550
C04803=1065.566,-74.686,-61.144,171.965,24.604,154.550
C04804=1065.560,-74.936,-61.132,171.963,24.603,154.550
C04805=1065.554,-75.186,-61.121,171.962,24.601,154.549
C04806=1065.548,-75.436,-61.110,171.959,24.599,154.549
C04807=1065.542,-75.685,-61.099,171.958,24.597,154.549
C04808=1065.536,-75.934,-61.088,171.956,24.596,154.549
C04809=1065.530,-76.184,-61.076,171.955,24.594,154.549
C04810=1065.524,-76.434,-61.066,171.953,24.592,154.549
C04811=1065.518,-76.684,-61.054,171.951,24.591,154.549
C04812=1065.512,-76.934,-61.043,171.950,24.589,154.549
C04813=1065.505,-77.183,-61.031,171.948,24.588,154.549
C04814=1065.500,-77.433,-61.021,171.947,24.586,154.549
C04815=1065.493,-77.683,-61.009,171.945,24.584,154.548
C04816=1065.488,-77.932,-60.998,171.943,24.583,154.548
C04817=1065.481,-78.181,-60.988,171.942,24.581,154.548
C04818=1065.475,-78.432,-60.977,171.940,24.580,154.548
C04819=1065.469,-78.681,-60.966,171.939,24.578,154.548
C04820=1065.463,-78.931,-60.955,171.937,24.576,154.548
C04821=1065.457,-79.180,-60.943,171.935,24.575,154.548
C04822=1065.451,-79.430,-60.932,171.934,24.573,154.548
C04823=1065.445,-79.680,-60.921,171.932,24.572,154.548
C04824=1065.439,-79.929,-60.910,171.931,24.570,154.548
C04825=1065.432,-80.180,-60.899,171.929,24.569,154.548
C04826=1065.426,-80.429,-60.889,171.927,24.567,154.547
C04827=1065.420,-80.678,-60.878,171.926,24.565,154.547
C04828=1065.414,-80.928,-60.867,171.923,24.563,154.547
C04829=1065.407,-81.178,-60.856,171.922,24.562,154.547
C04830=1065.401,-81.428,-60.845,171.920,24.560,154.547
C04831=1065.395,-81.677,-60.834,171.918,24.559,154.547
C04832=1065.388,-81.959,-60.822,171.917,24.557,154.547
C04833=1065.381,-82.240,-60.809,171.915,24.556,154.547
C04834=1065.374,-82.522,-60.797,171.913,24.554,154.547
C04835=1065.367,-82.803,-60.785,171.911,24.552,154.547
C04836=1065.361,-83.052,-60.774,171.909,24.551,154.547
C04837=1065.355,-83.301,-60.763,171.908,24.549,154.547
C04838=1065.349,-83.551,-60.752,171.906,24.548,154.547
C04839=1065.342,-83.801,-60.743,171.904,24.546,154.547
C04840=1065.337,-84.051,-60.732,171.903,24.545,154.546
C04841=1065.330,-84.301,-60.721,171.901,24.543,154.546
C04842=1065.324,-84.550,-60.710,171.900,24.542,154.546
C04843=1065.318,-84.800,-60.699,171.898,24.540,154.546
C04844=1065.312,-85.050,-60.688,171.896,24.539,154.546
C04845=1065.305,-85.299,-60.678,171.895,24.538,154.546
C04846=1065.299,-85.549,-60.667,171.893,24.536,154.546
C04847=1065.293,-85.799,-60.656,171.891,24.535,154.546
C04848=1065.287,-86.048,-60.645,171.890,24.533,154.546
C04849=1065.280,-86.298,-60.634,171.888,24.532,154.546
C04850=1065.275,-86.548,-60.624,171.887,24.530,154.546
C04851=1065.269,-86.797,-60.614,171.884,24.529,154.546
C04852=1065.262,-87.048,-60.603,171.882,24.527,154.546
C04853=1065.256,-87.297,-60.592,171.881,24.526,154.546
C04854=1065.250,-87.546,-60.581,171.879,24.524,154.546
C04855=1065.244,-87.796,-60.570,171.878,24.523,154.546
C04856=1065.238,-88.046,-60.559,171.876,24.521,154.546
C04857=1065.232,-88.296,-60.550,171.874,24.520,154.546
C04858=1065.226,-88.545,-60.539,171.873,24.518,154.545
C04859=1065.220,-88.795,-60.528,171.871,24.517,154.545
C04860=1065.213,-89.045,-60.517,171.869,24.516,154.545
C04861=1065.207,-89.294,-60.506,171.868,24.514,154.545
C04862=1065.202,-89.544,-60.496,171.866,24.513,154.545
C04863=1065.195,-89.794,-60.486,171.864,24.511,154.545
C04864=1065.189,-90.044,-60.475,171.863,24.510,154.545
C04865=1065.183,-90.293,-60.464,171.861,24.508,154.545
C04866=1065.177,-90.543,-60.454,171.859,24.507,154.545
C04867=1065.171,-90.793,-60.443,171.858,24.506,154.545
C04868=1065.164,-91.042,-60.433,171.856,24.505,154.545
C04869=1065.159,-91.292,-60.422,171.855,24.503,154.545
C04870=1065.153,-91.541,-60.412,171.853,24.501,154.545
C04871=1065.146,-91.792,-60.401,171.851,24.500,154.545
C04872=1065.140,-92.041,-60.390,171.849,24.499,154.545
C04873=1065.134,-92.291,-60.381,171.848,24.497,154.545
C04874=1065.129,-92.540,-60.370,171.846,24.496,154.545
C04875=1065.122,-92.790,-60.359,171.845,24.495,154.545
C04876=1065.116,-93.040,-60.348,171.843,24.493,154.545
C04877=1065.110,-93.290,-60.338,171.841,24.492,154.545
C04878=1065.104,-93.539,-60.328,171.839,24.490,154.545
C04879=1065.098,-93.789,-60.317,171.837,24.489,154.545
C04880=1065.092,-94.038,-60.307,171.835,24.487,154.545
C04881=1065.086,-94.289,-60.296,171.834,24.486,154.544
C04882=1065.080,-94.539,-60.286,171.832,24.485,154.544
C04883=1065.074,-94.788,-60.276,171.830,24.484,154.544
C04884=1065.068,-95.037,-60.265,171.829,24.482,154.544
C04885=1065.062,-95.287,-60.255,171.827,24.481,154.544
C04886=1065.056,-95.537,-60.244,171.825,24.479,154.544
C04887=1065.049,-95.787,-60.234,171.824,24.478,154.544
C04888=1065.044,-96.037,-60.223,171.822,24.477,154.544
C04889=1065.038,-96.286,-60.213,171.820,24.476,154.544
C04890=1065.032,-96.536,-60.203,171.819,24.474,154.544
C04891=1065.026,-96.785,-60.192,171.817,24.473,154.544
C04892=1065.020,-97.035,-60.183,171.815,24.471,154.544
C04893=1065.014,-97.285,-60.172,171.814,24.470,154.544
C04894=1065.007,-97.535,-60.161,171.812,24.469,154.544
C04895=1065.001,-97.785,-60.151,171.810,24.468,154.544
C04896=1064.994,-98.068,-60.139,171.809,24.466,154.544
C04897=1064.987,-98.351,-60.128,171.806,24.465,154.544
C04898=1064.980,-98.635,-60.116,171.804,24.463,154.544
C04899=1064.974,-98.919,-60.105,171.803,24.462,154.544
C04900=1064.967,-99.168,-60.094,171.801,24.461,154.544
C04901=1064.961,-99.418,-60.085,171.799,24.460,154.544
C04902=1064.955,-99.667,-60.074,171.798,24.458,154.544
C04903=1064.949,-99.917,-60.064,171.796,24.457,154.544
C04904=1064.942,-100.168,-60.054,171.794,24.456,154.544
C04905=1064.936,-100.417,-60.044,171.793,24.455,154.544
C04906=1064.930,-100.667,-60.034,171.791,24.453,154.544
C04907=1064.924,-100.916,-60.024,171.789,24.452,154.544
C04908=1064.918,-101.166,-60.014,171.788,24.451,154.544
C04909=1064.912,-101.415,-60.003,171.785,24.449,154.544
C04910=1064.906,-101.665,-59.994,171.783,24.448,154.544
C04911=1064.900,-101.915,-59.983,171.781,24.447,154.544
C04912=1064.893,-102.165,-59.973,171.780,24.446,154.544
C04913=1064.887,-102.415,-59.963,171.778,24.445,154.544
C04914=1064.881,-102.665,-59.952,171.776,24.444,154.544
C04915=1064.875,-102.914,-59.943,171.775,24.442,154.544
C04916=1064.869,-103.163,-59.933,171.773,24.441,154.544
C04917=1064.863,-103.414,-59.922,171.771,24.440,154.544
C04918=1064.857,-103.663,-59.913,171.770,24.439,154.544
C04919=1064.851,-103.913,-59.903,171.768,24.438,154.544
C04920=1064.844,-104.162,-59.893,171.766,24.437,154.544
C04921=1064.839,-104.412,-59.883,171.764,24.435,154.544
C04922=1064.832,-104.662,-59.873,171.763,24.434,154.544
C04923=1064.826,-104.911,-59.863,171.761,24.433,154.544
C04924=1064.820,-105.162,-59.852,171.759,24.432,154.544
C04925=1064.814,-105.411,-59.842,171.758,24.431,154.544
C04926=1064.808,-105.661,-59.833,171.756,24.430,154.544
C04927=1064.801,-105.911,-59.823,171.754,24.428,154.544
C04928=1064.796,-106.161,-59.812,171.753,24.427,154.544
C04929=1064.790,-106.410,-59.803,171.751,24.426,154.544
C04930=1064.783,-106.660,-59.793,171.749,24.425,154.544
C04931=1064.777,-106.910,-59.783,171.747,24.424,154.544
C04932=1064.771,-107.159,-59.773,171.746,24.423,154.544
C04933=1064.765,-107.409,-59.763,171.744,24.422,154.544
C04934=1064.759,-107.659,-59.753,171.742,24.421,154.544
C04935=1064.753,-107.909,-59.744,171.740,24.420,154.544
C04936=1064.746,-108.158,-59.734,171.739,24.419,154.544
C04937=1064.740,-108.408,-59.724,171.737,24.418,154.544
C04938=1064.734,-108.658,-59.714,171.735,24.416,154.544
C04939=1064.729,-108.908,-59.704,171.733,24.416,154.544
C04940=1064.723,-109.157,-59.695,171.732,24.414,154.544
C04941=1064.716,-109.407,-59.684,171.730,24.413,154.544
C04942=1064.710,-109.656,-59.675,171.728,24.412,154.544
C04943=1064.704,-109.906,-59.665,171.727,24.411,154.544
C04944=1064.698,-110.156,-59.656,171.725,24.410,154.544
C04945=1064.691,-110.406,-59.646,171.723,24.409,154.544
C04946=1064.685,-110.655,-59.636,171.721,24.408,154.544
C04947=1064.679,-110.905,-59.626,171.720,24.407,154.545
C04948=1064.673,-111.155,-59.617,171.718,24.406,154.545
C04949=1064.667,-111.405,-59.607,171.716,24.405,154.545
C04950=1064.661,-111.655,-59.597,171.714,24.404,154.545
C04951=1064.655,-111.904,-59.587,171.713,24.403,154.545
C04952=1064.649,-112.154,-59.578,171.711,24.402,154.545
C04953=1064.642,-112.404,-59.568,171.709,24.401,154.545
C04954=1064.636,-112.653,-59.558,171.707,24.400,154.545
C04955=1064.630,-112.903,-59.548,171.706,24.399,154.545
C04956=1064.624,-113.153,-59.539,171.704,24.398,154.545
C04957=1064.617,-113.402,-59.529,171.702,24.397,154.545
C04958=1064.611,-113.652,-59.520,171.700,24.396,154.545
C04959=1064.605,-113.902,-59.510,171.699,24.395,154.545
C04960=1064.599,-114.184,-59.499,171.696,24.394,154.545
C04961=1064.592,-114.466,-59.489,171.694,24.393,154.545
C04962=1064.584,-114.748,-59.478,171.692,24.392,154.545
C04963=1064.578,-115.029,-59.467,171.691,24.391,154.545
C04964=1064.572,-115.279,-59.458,171.689,24.390,154.545
C04965=1064.565,-115.528,-59.448,171.687,24.389,154.545
C04966=1064.559,-115.778,-59.439,171.685,24.388,154.545
C04967=1064.553,-116.028,-59.429,171.684,24.387,154.545
C04968=1064.547,-116.278,-59.420,171.682,24.386,154.545
C04969=1064.541,-116.528,-59.410,171.680,24.385,154.546
C04970=1064.535,-116.777,-59.400,171.678,24.384,154.546
C04971=1064.528,-117.027,-59.391,171.677,24.383,154.546
C04972=1064.522,-117.277,-59.381,171.675,24.383,154.546
C04973=1064.516,-117.527,-59.372,171.673,24.381,154.546
C04974=1064.510,-117.777,-59.362,171.671,24.381,154.546
C04975=1064.504,-118.026,-59.353,171.669,24.380,154.546
C04976=1064.498,-118.275,-59.343,171.668,24.379,154.546
C04977=1064.492,-118.525,-59.334,171.666,24.378,154.546
C04978=1064.486,-118.775,-59.324,171.664,24.377,154.546
C04979=1064.480,-119.025,-59.315,171.662,24.376,154.546
C04980=1064.473,-119.275,-59.305,171.661,24.375,154.546
C04981=1064.467,-119.524,-59.296,171.659,24.375,154.546
C04982=1064.460,-119.774,-59.287,171.657,24.373,154.546
C04983=1064.454,-120.024,-59.278,171.655,24.373,154.546
C04984=1064.448,-120.274,-59.268,171.653,24.372,154.547
C04985=1064.443,-120.523,-59.259,171.652,24.371,154.547
C04986=1064.437,-120.773,-59.249,171.650,24.370,154.547
C04987=1064.430,-121.023,-59.240,171.648,24.369,154.547
C04988=1064.424,-121.273,-59.230,171.646,24.369,154.547
C04989=1064.418,-121.522,-59.221,171.645,24.367,154.547
C04990=1064.411,-121.773,-59.212,171.643,24.367,154.547
C04991=1064.405,-122.022,-59.203,171.641,24.366,154.547
C04992=1064.400,-122.271,-59.194,171.639,24.365,154.547
C04993=1064.394,-122.521,-59.184,171.637,24.364,154.547
C04994=1064.387,-122.771,-59.175,171.635,24.364,154.547
C04995=1064.381,-123.021,-59.165,171.634,24.363,154.547
C04996=1064.375,-123.271,-59.157,171.632,24.362,154.548
C04997=1064.368,-123.521,-59.147,171.630,24.361,154.547
C04998=1064.363,-123.770,-59.138,171.628,24.360,154.548
C04999=1064.357,-124.020,-59.128,171.626,24.360,154.548
C05000=1064.351,-124.270,-59.120,171.625,24.359,154.548
C05001=1064.345,-124.520,-59.110,171.623,24.358,154.548
C05002=1064.338,-124.769,-59.101,171.621,24.357,154.548
C05003=1064.332,-125.018,-59.092,171.619,24.356,154.548
C05004=1064.326,-125.269,-59.083,171.617,24.356,154.548
C05005=1064.320,-125.519,-59.073,171.616,24.355,154.548
C05006=1064.313,-125.768,-59.064,171.614,24.354,154.548
C05007=1064.307,-126.018,-59.055,171.612,24.354,154.548
C05008=1064.301,-126.268,-59.046,171.610,24.353,154.549
C05009=1064.295,-126.517,-59.037,171.608,24.352,154.549
C05010=1064.289,-126.767,-59.028,171.606,24.351,154.549
C05011=1064.283,-127.017,-59.019,171.605,24.351,154.549
C05012=1064.277,-127.267,-59.009,171.603,24.350,154.549
C05013=1064.270,-127.516,-59.001,171.601,24.349,154.549
C05014=1064.264,-127.766,-58.991,171.599,24.348,154.549
C05015=1064.258,-128.016,-58.982,171.597,24.348,154.549
C05016=1064.255,-128.267,-58.972,171.596,24.346,154.549
C05017=1064.253,-128.518,-58.961,171.594,24.344,154.549
C05018=1064.252,-128.768,-58.949,171.593,24.341,154.549
C05019=1064.253,-129.018,-58.938,171.592,24.337,154.548
C05020=1064.255,-129.271,-58.923,171.592,24.333,154.547
C05021=1064.259,-129.522,-58.910,171.591,24.329,154.547
C05022=1064.265,-129.774,-58.895,171.591,24.323,154.546
C05023=1064.272,-130.023,-58.880,171.590,24.317,154.545
C05024=1063.888,-130.046,-59.062,171.544,24.469,154.578
C05025=1063.881,-129.796,-59.077,171.543,24.474,154.579
C05026=1063.875,-129.545,-59.092,171.544,24.479,154.579
C05027=1063.871,-129.293,-59.107,171.545,24.484,154.580
C05028=1063.869,-129.041,-59.120,171.546,24.488,154.581
C05029=1063.868,-128.791,-59.132,171.546,24.492,154.581
C05030=1063.869,-128.540,-59.145,171.547,24.495,154.582
C05031=1063.871,-128.289,-59.155,171.548,24.497,154.582
C05032=1063.875,-128.039,-59.165,171.550,24.499,154.582
C05033=1063.880,-127.789,-59.175,171.552,24.499,154.582
C05034=1063.885,-127.539,-59.184,171.554,24.500,154.582
C05035=1063.892,-127.290,-59.193,171.555,24.501,154.582
C05036=1063.899,-127.040,-59.202,171.557,24.501,154.582
C05037=1063.904,-126.789,-59.211,171.559,24.502,154.582
C05038=1063.911,-126.540,-59.220,171.561,24.503,154.582
C05039=1063.917,-126.291,-59.229,171.563,24.504,154.582
C05040=1063.923,-126.040,-59.238,171.564,24.505,154.581
C05041=1063.929,-125.791,-59.248,171.566,24.505,154.581
C05042=1063.936,-125.541,-59.257,171.568,24.506,154.581
C05043=1063.942,-125.291,-59.266,171.570,24.507,154.581
C05044=1063.947,-125.042,-59.275,171.572,24.507,154.581
C05045=1063.953,-124.792,-59.284,171.574,24.508,154.581
C05046=1063.960,-124.542,-59.293,171.575,24.509,154.581
C05047=1063.967,-124.293,-59.303,171.577,24.510,154.581
C05048=1063.972,-124.042,-59.312,171.579,24.511,154.581
C05049=1063.979,-123.792,-59.321,171.581,24.511,154.581
C05050=1063.984,-123.543,-59.330,171.583,24.512,154.580
C05051=1063.991,-123.294,-59.339,171.584,24.513,154.580
C05052=1063.997,-123.044,-59.349,171.586,24.514,154.580
C05053=1064.003,-122.794,-59.358,171.588,24.515,154.580
C05054=1064.009,-122.544,-59.367,171.590,24.515,154.580
C05055=1064.015,-122.294,-59.377,171.592,24.516,154.580
C05056=1064.021,-122.045,-59.386,171.593,24.517,154.580
C05057=1064.028,-121.795,-59.395,171.595,24.518,154.580
C05058=1064.034,-121.545,-59.404,171.597,24.519,154.580
C05059=1064.040,-121.295,-59.414,171.599,24.519,154.580
C05060=1064.046,-121.045,-59.423,171.601,24.520,154.580
C05061=1064.052,-120.796,-59.433,171.602,24.521,154.580
C05062=1064.058,-120.546,-59.442,171.604,24.522,154.579
C05063=1064.064,-120.297,-59.452,171.606,24.522,154.579
C05064=1064.070,-120.047,-59.461,171.608,24.524,154.579
C05065=1064.076,-119.797,-59.471,171.610,24.524,154.579
C05066=1064.083,-119.547,-59.479,171.611,24.525,154.579
C05067=1064.089,-119.297,-59.488,171.613,24.526,154.579
C05068=1064.095,-119.047,-59.498,171.615,24.527,154.579
C05069=1064.102,-118.798,-59.508,171.617,24.528,154.579
C05070=1064.108,-118.548,-59.517,171.618,24.529,154.579
C05071=1064.113,-118.299,-59.526,171.620,24.530,154.579
C05072=1064.119,-118.049,-59.536,171.622,24.530,154.579
C05073=1064.126,-117.799,-59.546,171.624,24.532,154.579
C05074=1064.132,-117.549,-59.555,171.626,24.532,154.579
C05075=1064.138,-117.299,-59.565,171.627,24.533,154.579
C05076=1064.144,-117.050,-59.574,171.629,24.534,154.579
C05077=1064.150,-116.800,-59.584,171.631,24.535,154.578
C05078=1064.156,-116.550,-59.593,171.633,24.536,154.578
C05079=1064.163,-116.300,-59.603,171.635,24.537,154.578
C05080=1064.170,-116.051,-59.612,171.636,24.538,154.578
C05081=1064.176,-115.801,-59.621,171.638,24.539,154.578
C05082=1064.182,-115.551,-59.631,171.640,24.539,154.578
C05083=1064.188,-115.301,-59.641,171.642,24.541,154.578
C05084=1064.194,-115.052,-59.650,171.643,24.541,154.578
C05085=1064.200,-114.770,-59.661,171.645,24.542,154.578
C05086=1064.208,-114.488,-59.672,171.648,24.543,154.578
C05087=1064.215,-114.206,-59.683,171.650,24.545,154.578
C05088=1064.221,-113.925,-59.694,171.651,24.546,154.578
C05089=1064.227,-113.675,-59.703,171.653,24.547,154.578
C05090=1064.233,-113.425,-59.713,171.655,24.548,154.578
C05091=1064.239,-113.175,-59.722,171.657,24.549,154.578
C05092=1064.245,-112.925,-59.732,171.658,24.550,154.578
C05093=1064.252,-112.676,-59.741,171.660,24.550,154.578
C05094=1064.258,-112.426,-59.751,171.662,24.552,154.578
C05095=1064.264,-112.177,-59.761,171.664,24.552,154.578
C05096=1064.270,-111.927,-59.771,171.665,24.554,154.578
C05097=1064.277,-111.677,-59.780,171.667,24.554,154.577
C05098=1064.283,-111.427,-59.790,171.669,24.556,154.577
C05099=1064.288,-111.177,-59.800,171.671,24.557,154.578
C05100=1064.294,-110.927,-59.810,171.672,24.557,154.577
C05101=1064.301,-110.677,-59.819,171.674,24.559,154.577
C05102=1064.307,-110.428,-59.829,171.676,24.559,154.577
C05103=1064.313,-110.179,-59.839,171.678,24.561,154.577
C05104=1064.319,-109.929,-59.849,171.679,24.562,154.577
C05105=1064.326,-109.679,-59.858,171.681,24.563,154.577
C05106=1064.332,-109.429,-59.868,171.683,24.564,154.577
C05107=1064.338,-109.179,-59.877,171.684,24.565,154.577
C05108=1064.344,-108.930,-59.888,171.686,24.566,154.577
C05109=1064.350,-108.680,-59.898,171.688,24.567,154.577
C05110=1064.356,-108.430,-59.907,171.691,24.569,154.577
C05111=1064.362,-108.180,-59.917,171.692,24.569,154.577
C05112=1064.369,-107.931,-59.927,171.694,24.570,154.577
C05113=1064.375,-107.681,-59.937,171.696,24.572,154.577
C05114=1064.381,-107.432,-59.946,171.698,24.572,154.577
C05115=1064.386,-107.182,-59.956,171.699,24.574,154.577
C05116=1064.393,-106.932,-59.967,171.701,24.575,154.577
C05117=1064.399,-106.683,-59.976,171.703,24.576,154.577
C05118=1064.405,-106.433,-59.986,171.705,24.577,154.577
C05119=1064.412,-106.182,-59.996,171.706,24.578,154.577
C05120=1064.418,-105.933,-60.007,171.708,24.579,154.577
C05121=1064.424,-105.683,-60.016,171.710,24.581,154.577
C05122=1064.430,-105.433,-60.026,171.711,24.581,154.577
C05123=1064.437,-105.184,-60.036,171.713,24.582,154.577
C05124=1064.442,-104.934,-60.046,171.715,24.584,154.577
C05125=1064.448,-104.684,-60.056,171.717,24.585,154.577
C05126=1064.455,-104.435,-60.066,171.718,24.586,154.577
C05127=1064.460,-104.185,-60.076,171.720,24.587,154.577
C05128=1064.466,-103.935,-60.086,171.722,24.588,154.577
C05129=1064.473,-103.686,-60.096,171.723,24.589,154.577
C05130=1064.479,-103.436,-60.106,171.725,24.591,154.577
C05131=1064.484,-103.186,-60.116,171.727,24.592,154.577
C05132=1064.491,-102.937,-60.126,171.729,24.593,154.577
C05133=1064.497,-102.687,-60.136,171.730,24.594,154.577
C05134=1064.503,-102.437,-60.147,171.732,24.595,154.577
C05135=1064.510,-102.187,-60.157,171.734,24.596,154.577
C05136=1064.516,-101.937,-60.166,171.735,24.598,154.577
C05137=1064.521,-101.688,-60.177,171.737,24.599,154.577
C05138=1064.528,-101.438,-60.187,171.739,24.600,154.577
C05139=1064.534,-101.189,-60.197,171.740,24.601,154.577
C05140=1064.540,-100.939,-60.207,171.742,24.603,154.577
C05141=1064.546,-100.689,-60.217,171.744,24.604,154.577
C05142=1064.553,-100.439,-60.227,171.746,24.605,154.577
C05143=1064.558,-100.189,-60.237,171.747,24.606,154.577
C05144=1064.565,-99.940,-60.248,171.749,24.607,154.577
C05145=1064.571,-99.690,-60.257,171.751,24.608,154.577
C05146=1064.577,-99.440,-60.268,171.752,24.609,154.577
C05147=1064.583,-99.191,-60.278,171.754,24.611,154.577
C05148=1064.589,-98.941,-60.288,171.756,24.612,154.577
C05149=1064.596,-98.657,-60.300,171.758,24.614,154.577
C05150=1064.603,-98.374,-60.312,171.760,24.615,154.577
C05151=1064.611,-98.089,-60.323,171.762,24.617,154.577
C05152=1064.617,-97.806,-60.335,171.764,24.618,154.577
C05153=1064.623,-97.556,-60.345,171.766,24.619,154.577
C05154=1064.630,-97.307,-60.355,171.768,24.621,154.577
C05155=1064.635,-97.057,-60.365,171.769,24.622,154.577
C05156=1064.641,-96.808,-60.376,171.771,24.623,154.577
C05157=1064.648,-96.557,-60.386,171.773,24.624,154.577
C05158=1064.653,-96.308,-60.397,171.774,24.626,154.577
C05159=1064.660,-96.058,-60.407,171.776,24.627,154.577
C05160=1064.665,-95.808,-60.417,171.778,24.628,154.577
C05161=1064.672,-95.559,-60.428,171.779,24.630,154.577
C05162=1064.677,-95.309,-60.438,171.781,24.631,154.577
C05163=1064.684,-95.059,-60.448,171.783,24.632,154.577
C05164=1064.690,-94.810,-60.459,171.784,24.634,154.577
C05165=1064.695,-94.560,-60.469,171.786,24.635,154.577
C05166=1064.702,-94.310,-60.480,171.788,24.636,154.577
C05167=1064.708,-94.061,-60.491,171.789,24.638,154.577
C05168=1064.714,-93.811,-60.500,171.791,24.639,154.577
C05169=1064.720,-93.561,-60.511,171.793,24.640,154.577
C05170=1064.726,-93.311,-60.522,171.794,24.642,154.577
C05171=1064.732,-93.062,-60.532,171.796,24.643,154.578
C05172=1064.738,-92.812,-60.543,171.798,24.645,154.578
C05173=1064.744,-92.563,-60.553,171.799,24.646,154.578
C05174=1064.750,-92.312,-60.564,171.801,24.647,154.578
C05175=1064.757,-92.063,-60.574,171.803,24.649,154.578
C05176=1064.763,-91.813,-60.585,171.804,24.650,154.578
C05177=1064.768,-91.563,-60.595,171.807,24.652,154.578
C05178=1064.774,-91.314,-60.605,171.809,24.653,154.578
C05179=1064.781,-91.064,-60.616,171.810,24.654,154.578
C05180=1064.787,-90.814,-60.627,171.812,24.656,154.578
C05181=1064.793,-90.565,-60.637,171.813,24.657,154.578
C05182=1064.798,-90.315,-60.648,171.815,24.659,154.578
C05183=1064.806,-90.065,-60.658,171.817,24.660,154.578
C05184=1064.811,-89.816,-60.669,171.819,24.661,154.578
C05185=1064.817,-89.566,-60.679,171.820,24.663,154.578
C05186=1064.823,-89.317,-60.690,171.822,24.664,154.578
C05187=1064.830,-89.066,-60.701,171.823,24.666,154.578
C05188=1064.835,-88.817,-60.712,171.825,24.667,154.578
C05189=1064.842,-88.568,-60.722,171.827,24.669,154.578
C05190=1064.848,-88.317,-60.733,171.828,24.670,154.578
C05191=1064.854,-88.068,-60.743,171.830,24.671,154.578
C05192=1064.860,-87.818,-60.754,171.832,24.673,154.579
C05193=1064.866,-87.568,-60.765,171.833,24.674,154.579
C05194=1064.873,-87.319,-60.775,171.835,24.675,154.579
C05195=1064.879,-87.069,-60.786,171.837,24.677,154.579
C05196=1064.884,-86.820,-60.797,171.838,24.678,154.579
C05197=1064.891,-86.569,-60.807,171.840,24.680,154.579
C05198=1064.897,-86.320,-60.818,171.841,24.682,154.579
C05199=1064.903,-86.070,-60.829,171.843,24.683,154.579
C05200=1064.910,-85.820,-60.839,171.845,24.684,154.579
C05201=1064.915,-85.571,-60.850,171.846,24.686,154.579
C05202=1064.921,-85.321,-60.861,171.849,24.687,154.579
C05203=1064.928,-85.072,-60.872,171.851,24.689,154.579
C05204=1064.934,-84.822,-60.883,171.852,24.690,154.579
C05205=1064.940,-84.573,-60.894,171.854,24.692,154.579
C05206=1064.947,-84.323,-60.904,171.856,24.694,154.579
C05207=1064.952,-84.073,-60.915,171.857,24.695,154.579
C05208=1064.959,-83.822,-60.926,171.859,24.696,154.579
C05209=1064.964,-83.573,-60.936,171.860,24.698,154.580
C05210=1064.971,-83.324,-60.947,171.862,24.699,154.580
C05211=1064.977,-83.074,-60.958,171.864,24.701,154.580
C05212=1064.983,-82.824,-60.969,171.865,24.702,154.580
C05213=1064.990,-82.543,-60.982,171.867,24.704,154.580
C05214=1064.997,-82.261,-60.994,171.870,24.706,154.580
C05215=1065.004,-81.980,-61.006,171.871,24.707,154.580
C05216=1065.012,-81.699,-61.018,171.873,24.709,154.580
C05217=1065.017,-81.450,-61.029,171.874,24.710,154.580
C05218=1065.024,-81.199,-61.040,171.876,24.712,154.580
C05219=1065.030,-80.950,-61.051,171.878,24.713,154.580
C05220=1065.037,-80.700,-61.062,171.879,24.715,154.580
C05221=1065.042,-80.451,-61.072,171.881,24.717,154.580
C05222=1065.048,-80.201,-61.083,171.882,24.718,154.580
C05223=1065.054,-79.951,-61.095,171.885,24.720,154.581
C05224=1065.061,-79.702,-61.105,171.887,24.721,154.581
C05225=1065.067,-79.451,-61.116,171.888,24.723,154.581
C05226=1065.073,-79.202,-61.127,171.890,24.724,154.581
C05227=1065.079,-78.952,-61.138,171.891,24.726,154.581
C05228=1065.085,-78.702,-61.149,171.893,24.728,154.581
C05229=1065.091,-78.453,-61.160,171.895,24.729,154.581
C05230=1065.097,-78.203,-61.172,171.896,24.731,154.581
C05231=1065.103,-77.954,-61.183,171.898,24.732,154.581
C05232=1065.110,-77.704,-61.194,171.899,24.734,154.581
C05233=1065.115,-77.454,-61.205,171.901,24.736,154.581
C05234=1065.121,-77.205,-61.216,171.903,24.737,154.581
C05235=1065.127,-76.954,-61.227,171.904,24.739,154.582
C05236=1065.134,-76.705,-61.237,171.906,24.741,154.582
C05237=1065.140,-76.456,-61.249,171.907,24.742,154.582
C05238=1065.146,-76.206,-61.260,171.909,24.744,154.582
C05239=1065.153,-75.956,-61.271,171.911,24.746,154.582
C05240=1065.158,-75.706,-61.282,171.912,24.747,154.582
C05241=1065.164,-75.457,-61.293,171.914,24.749,154.582
C05242=1065.171,-75.207,-61.305,171.915,24.750,154.582
C05243=1065.176,-74.958,-61.316,171.917,24.752,154.582
C05244=1065.183,-74.708,-61.327,171.919,24.753,154.583
C05245=1065.188,-74.458,-61.338,171.921,24.756,154.583
C05246=1065.195,-74.209,-61.350,171.923,24.757,154.583
C05247=1065.201,-73.959,-61.361,171.924,24.759,154.583
C05248=1065.207,-73.709,-61.372,171.926,24.760,154.583
C05249=1065.213,-73.459,-61.383,171.927,24.762,154.583
C05250=1065.220,-73.210,-61.395,171.929,24.764,154.583
C05251=1065.225,-72.960,-61.406,171.931,24.765,154.583
C05252=1065.230,-72.711,-61.417,171.932,24.767,154.583
C05253=1065.237,-72.460,-61.429,171.934,24.769,154.583
C05254=1065.243,-72.212,-61.440,171.935,24.771,154.584
C05255=1065.249,-71.961,-61.451,171.937,24.773,154.584
C05256=1065.254,-71.712,-61.463,171.938,24.774,154.584
C05257=1065.261,-71.462,-61.475,171.940,24.776,154.584
C05258=1065.266,-71.213,-61.486,171.942,24.777,154.584
C05259=1065.273,-70.962,-61.497,171.943,24.779,154.584
C05260=1065.279,-70.713,-61.509,171.945,24.781,154.584
C05261=1065.284,-70.463,-61.520,171.946,24.783,154.584
C05262=1065.290,-70.213,-61.531,171.948,24.785,154.585
C05263=1065.297,-69.964,-61.543,171.949,24.787,154.585
C05264=1065.303,-69.714,-61.554,171.951,24.788,154.585
C05265=1065.309,-69.465,-61.566,171.953,24.790,154.585
C05266=1065.314,-69.215,-61.578,171.955,24.792,154.585
C05267=1065.321,-68.965,-61.589,171.957,24.794,154.585
C05268=1065.327,-68.716,-61.600,171.958,24.795,154.585
C05269=1065.333,-68.466,-61.612,171.960,24.797,154.585
C05270=1065.339,-68.217,-61.623,171.961,24.799,154.586
C05271=1065.345,-67.966,-61.635,171.963,24.801,154.586
C05272=1065.351,-67.718,-61.647,171.964,24.803,154.586
C05273=1065.357,-67.467,-61.658,171.966,24.804,154.586
C05274=1065.363,-67.218,-61.669,171.968,24.806,154.586
C05275=1065.369,-66.968,-61.681,171.969,24.808,154.586
C05276=1065.374,-66.718,-61.692,171.971,24.810,154.586
C05277=1065.382,-66.439,-61.706,171.972,24.812,154.587
C05278=1065.388,-66.160,-61.719,171.975,24.814,154.587
C05279=1065.396,-65.881,-61.731,171.976,24.816,154.587
C05280=1065.402,-65.602,-61.744,171.978,24.818,154.587
C05281=1065.407,-65.352,-61.756,171.979,24.820,154.587
C05282=1065.414,-65.102,-61.768,171.981,24.822,154.587
C05283=1065.420,-64.853,-61.779,171.982,24.823,154.588
C05284=1065.426,-64.603,-61.791,171.984,24.825,154.588
C05285=1065.432,-64.354,-61.803,171.985,24.827,154.588
C05286=1065.438,-64.104,-61.814,171.987,24.829,154.588
C05287=1065.445,-63.854,-61.826,171.988,24.831,154.588
C05288=1065.450,-63.605,-61.837,171.991,24.833,154.588
C05289=1065.456,-63.355,-61.849,171.993,24.835,154.588
C05290=1065.462,-63.105,-61.860,171.994,24.836,154.588
C05291=1065.469,-62.856,-61.872,171.996,24.838,154.589
C05292=1065.475,-62.606,-61.884,171.997,24.840,154.589
C05293=1065.480,-62.356,-61.896,171.999,24.842,154.589
C05294=1065.487,-62.107,-61.908,172.000,24.844,154.589
C05295=1065.493,-61.856,-61.919,172.002,24.845,154.589
C05296=1065.499,-61.607,-61.931,172.003,24.847,154.589
C05297=1065.505,-61.358,-61.943,172.005,24.849,154.589
C05298=1065.511,-61.108,-61.954,172.006,24.851,154.590
C05299=1065.517,-60.858,-61.967,172.008,24.853,154.590
C05300=1065.524,-60.609,-61.978,172.010,24.855,154.590
C05301=1065.529,-60.359,-61.989,172.011,24.856,154.590
C05302=1065.536,-60.110,-62.001,172.013,24.858,154.590
C05303=1065.542,-59.860,-62.014,172.014,24.860,154.590
C05304=1065.548,-59.610,-62.025,172.016,24.862,154.590
C05305=1065.554,-59.361,-62.037,172.017,24.864,154.591
C05306=1065.560,-59.111,-62.049,172.019,24.866,154.591
C05307=1065.567,-58.861,-62.060,172.020,24.868,154.591
C05308=1065.573,-58.612,-62.072,172.022,24.870,154.591
C05309=1065.579,-58.362,-62.085,172.024,24.872,154.591
C05310=1065.585,-58.112,-62.097,172.026,24.874,154.591
C05311=1065.591,-57.863,-62.107,172.027,24.875,154.592
C05312=1065.597,-57.613,-62.120,172.029,24.877,154.592
C05313=1065.603,-57.363,-62.132,172.031,24.879,154.592
C05314=1065.610,-57.114,-62.144,172.032,24.881,154.592
C05315=1065.615,-56.864,-62.155,172.034,24.883,154.592
C05316=1065.622,-56.614,-62.167,172.035,24.885,154.592
C05317=1065.628,-56.365,-62.179,172.037,24.887,154.593
C05318=1065.634,-56.115,-62.192,172.038,24.889,154.593
C05319=1065.640,-55.866,-62.203,172.040,24.890,154.593
C05320=1065.646,-55.616,-62.215,172.041,24.892,154.593
C05321=1065.653,-55.366,-62.227,172.043,24.894,154.593
C05322=1065.659,-55.116,-62.239,172.044,24.896,154.593
C05323=1065.665,-54.867,-62.251,172.046,24.898,154.594
C05324=1065.671,-54.618,-62.263,172.047,24.900,154.594
C05325=1065.678,-54.368,-62.275,172.049,24.902,154.594
C05326=1065.683,-54.118,-62.287,172.051,24.904,154.594
C05327=1065.690,-53.869,-62.299,172.052,24.905,154.594
C05328=1065.696,-53.619,-62.311,172.054,24.907,154.594
C05329=1065.702,-53.369,-62.323,172.056,24.909,154.594
C05330=1065.709,-53.120,-62.335,172.058,24.912,154.595
C05331=1065.715,-52.870,-62.348,172.059,24.914,154.595
C05332=1065.721,-52.620,-62.359,172.061,24.915,154.595
C05333=1065.727,-52.371,-62.371,172.062,24.917,154.595
C05334=1065.733,-52.121,-62.383,172.064,24.919,154.595
C05335=1065.740,-51.871,-62.395,172.065,24.921,154.595
C05336=1065.745,-51.621,-62.408,172.067,24.923,154.596
C05337=1065.752,-51.372,-62.420,172.068,24.925,154.596
C05338=1065.758,-51.123,-62.431,172.070,24.927,154.596
C05339=1065.764,-50.873,-62.444,172.071,24.929,154.596
C05340=1065.771,-50.624,-62.456,172.073,24.931,154.596
C05341=1065.777,-50.345,-62.469,172.074,24.933,154.596
C05342=1065.784,-50.068,-62.483,172.077,24.935,154.597
C05343=1065.791,-49.789,-62.497,172.078,24.937,154.597
C05344=1065.798,-49.511,-62.511,172.080,24.940,154.597
C05345=1065.804,-49.263,-62.523,172.081,24.941,154.597
C05346=1065.810,-49.013,-62.535,172.083,24.944,154.597
C05347=1065.816,-48.763,-62.548,172.084,24.946,154.598
C05348=1065.822,-48.513,-62.560,172.086,24.948,154.598
C05349=1065.828,-48.264,-62.572,172.087,24.950,154.598
C05350=1065.833,-48.014,-62.584,172.089,24.952,154.598
C05351=1065.839,-47.764,-62.597,172.090,24.954,154.598
C05352=1065.846,-47.515,-62.609,172.092,24.956,154.599
C05353=1065.852,-47.265,-62.621,172.094,24.958,154.599
C05354=1065.857,-47.016,-62.634,172.096,24.960,154.599
C05355=1065.864,-46.766,-62.646,172.097,24.963,154.599
C05356=1065.870,-46.516,-62.658,172.099,24.964,154.599
C05357=1065.876,-46.266,-62.671,172.100,24.966,154.599
C05358=1065.882,-46.016,-62.683,172.102,24.969,154.600
C05359=1065.889,-45.767,-62.696,172.103,24.970,154.600
C05360=1065.894,-45.518,-62.708,172.105,24.973,154.600
C05361=1065.900,-45.268,-62.721,172.106,24.975,154.600
C05362=1065.906,-45.019,-62.733,172.108,24.977,154.601
C05363=1065.912,-44.769,-62.745,172.109,24.979,154.601
C05364=1065.918,-44.519,-62.758,172.111,24.981,154.601
C05365=1065.924,-44.269,-62.770,172.112,24.983,154.601
C05366=1065.931,-44.020,-62.783,172.113,24.985,154.601
C05367=1065.937,-43.770,-62.796,172.115,24.987,154.602
C05368=1065.942,-43.521,-62.808,172.117,24.989,154.602
C05369=1065.948,-43.271,-62.820,172.118,24.991,154.602
C05370=1065.955,-43.022,-62.832,172.120,24.993,154.602
C05371=1065.961,-42.772,-62.845,172.121,24.995,154.602
C05372=1065.967,-42.523,-62.858,172.123,24.997,154.603
C05373=1065.973,-42.273,-62.871,172.124,25.000,154.603
C05374=1065.980,-42.023,-62.883,172.126,25.001,154.603
C05375=1065.985,-41.773,-62.895,172.127,25.004,154.603
C05376=1065.992,-41.524,-62.908,172.129,25.006,154.603
C05377=1065.998,-41.274,-62.921,172.131,25.008,154.604
C05378=1066.004,-41.025,-62.933,172.132,25.010,154.604
C05379=1066.010,-40.775,-62.945,172.134,25.012,154.604
C05380=1066.016,-40.526,-62.958,172.135,25.014,154.604
C05381=1066.022,-40.276,-62.971,172.137,25.017,154.604
C05382=1066.028,-40.026,-62.983,172.138,25.018,154.605
C05383=1066.034,-39.777,-62.995,172.140,25.021,154.605
C05384=1066.040,-39.527,-63.009,172.141,25.023,154.605
C05385=1066.046,-39.278,-63.021,172.143,25.025,154.605
C05386=1066.052,-39.028,-63.034,172.144,25.027,154.605
C05387=1066.059,-38.779,-63.046,172.146,25.029,154.606
C05388=1066.065,-38.529,-63.059,172.147,25.031,154.606
C05389=1066.071,-38.279,-63.072,172.149,25.033,154.606
C05390=1066.077,-38.030,-63.085,172.150,25.036,154.606
C05391=1066.083,-37.780,-63.097,172.152,25.038,154.607
C05392=1066.089,-37.530,-63.110,172.153,25.040,154.607
C05393=1066.095,-37.281,-63.123,172.155,25.042,154.607
C05394=1066.101,-37.031,-63.136,172.156,25.045,154.607
C05395=1066.107,-36.782,-63.149,172.158,25.046,154.607
C05396=1066.113,-36.532,-63.162,172.159,25.049,154.608
C05397=1066.119,-36.282,-63.174,172.160,25.051,154.608
C05398=1066.125,-36.033,-63.187,172.162,25.053,154.608
C05399=1066.131,-35.783,-63.200,172.163,25.055,154.608
C05400=1066.137,-35.534,-63.213,172.165,25.058,154.609
C05401=1066.143,-35.284,-63.225,172.166,25.059,154.609
C05402=1066.149,-35.034,-63.238,172.168,25.062,154.609
C05403=1066.155,-34.785,-63.251,172.169,25.064,154.609
C05404=1066.161,-34.535,-63.264,172.172,25.066,154.609
C05405=1066.168,-34.258,-63.279,172.173,25.069,154.610
C05406=1066.174,-33.980,-63.293,172.175,25.071,154.610
C05407=1066.181,-33.702,-63.308,172.176,25.073,154.610
C05408=1066.188,-33.425,-63.322,172.178,25.076,154.610
C05409=1066.194,-33.175,-63.335,172.180,25.078,154.611
C05410=1066.200,-32.925,-63.348,172.181,25.081,154.611
C05411=1066.206,-32.676,-63.361,172.183,25.083,154.611
C05412=1066.212,-32.426,-63.373,172.184,25.085,154.611
C05413=1066.219,-32.177,-63.387,172.186,25.087,154.612
C05414=1066.224,-31.927,-63.399,172.187,25.090,154.612
C05415=1066.231,-31.678,-63.413,172.189,25.092,154.612
C05416=1066.237,-31.428,-63.425,172.190,25.094,154.612
C05417=1066.243,-31.179,-63.438,172.191,25.096,154.613
C05418=1066.249,-30.930,-63.452,172.193,25.099,154.613
C05419=1066.255,-30.680,-63.464,172.194,25.100,154.613
C05420=1066.261,-30.430,-63.477,172.196,25.103,154.613
C05421=1066.267,-30.180,-63.490,172.197,25.105,154.614
C05422=1066.273,-29.931,-63.504,172.199,25.107,154.614
C05423=1066.278,-29.681,-63.516,172.200,25.109,154.614
C05424=1066.285,-29.432,-63.530,172.202,25.112,154.614
C05425=1066.291,-29.182,-63.543,172.203,25.114,154.615
C05426=1066.297,-28.932,-63.556,172.205,25.116,154.615
C05427=1066.304,-28.683,-63.569,172.206,25.118,154.615
C05428=1066.310,-28.433,-63.582,172.208,25.121,154.615
C05429=1066.316,-28.184,-63.595,172.209,25.123,154.615
C05430=1066.322,-27.934,-63.608,172.210,25.125,154.616
C05431=1066.328,-27.685,-63.622,172.212,25.127,154.616
C05432=1066.334,-27.435,-63.634,172.213,25.129,154.616
C05433=1066.340,-27.186,-63.647,172.215,25.132,154.616
C05434=1066.347,-26.936,-63.661,172.216,25.134,154.617
C05435=1066.352,-26.686,-63.674,172.218,25.136,154.617
C05436=1066.358,-26.436,-63.687,172.219,25.138,154.617
C05437=1066.365,-26.187,-63.701,172.221,25.141,154.617
C05438=1066.371,-25.937,-63.713,172.223,25.143,154.618
C05439=1066.376,-25.688,-63.727,172.225,25.146,154.618
C05440=1066.382,-25.438,-63.740,172.226,25.148,154.618
